# B&R Automation Studio project CombinedLinenSoiledA9KAN (part 3)

#### 6_sdc1Cyclic.ab
```automation-basic
PROGRAM _CYCLIC
	(* cyclic program *)

;Sequence 6 - Discharger 1 D[906]
a

;-----------------------------------------
;Revision 1.00 19/12/2005 D.J. First Issue
;-----------------------------------------

DischargerEnable 		= ((D[17] > 0) AND NOT Std.HaltSys)

I_BagAtBuffer			  = X[3].X06
I_BagAtDischarger	= X[3].X05
I_BagEmpty        = X[6].X01

I_OpenBag				= CAN[2].DropLoad OR TestDrop           ;X[23].X01
I_LoadDropped			= CAN[2].LoadDropped OR TestDischarger  ;X[23].X02

O_Steadys				= FALSE ;Y[6].Y01
O_OpenBuffer 			= FALSE ;Y[6].Y02
O_OpenBag				= FALSE ;Y[6].Y03
O_OpenStop				= FALSE ;Y[6].Y04
O_Closer				= FALSE ;Y[6].Y05

;Alarm
Alarm[7].Name 			= 0 ;Clear sequence alarm name
Alarm[7].Bag 			= 231
Alarm[7].Beacon			= TRUE
Alarm[7].Extra			= 0
Alarm[7].Time			= 3000

;Setup Sequence
STEP = D[907]
;Setup Pulse contact
PLS = (STEP <> LASTSTEP)
LASTSTEP = STEP

;Step 0 - Disabled
IF (STEP = 0) THEN
	;Disabled
ENDIF

;Check Status - Bag settled at buffer, no bag at discharger, bag at buffer on screen and no bag at discharger on the screen
TON_10ms(I_BagAtBuffer,300,SettledAtBuffer,SettledAtBufferET)
IF (STEP = 1) THEN
	IF (DischargerEnable AND SettledAtBuffer AND NOT I_BagAtDischarger AND (Bag[231].Cat = 0) AND NOT Std.HaltSys) THEN
		D[907] = 2
	ENDIF
	IF (Bag[231].Cat > 0) THEN
		Alarm[7].Name = almBagDataError
	ELSE IF I_BagAtDischarger THEN
		Alarm[7].Name = almSwitchFault
	ENDIF
ENDIF

;Wait for bag in discharger
IF (STEP = 2) THEN
	O_OpenBuffer 	= TRUE
	;Enable.SDC[1] 	= TRUE
	IF I_BagAtDischarger THEN
		D[907] = 3
	ENDIF
	Alarm[7].Name = almBagNotArrived
ENDIF

;Let bag settle in discharger
TON_10ms(((STEP = 3) AND I_BagAtDischarger),1000,SettledAtDischarger,SettledAtDischargerET)
IF (STEP = 3) THEN
	IF (Bag[231].Cat = 0) AND (Bag[229].Cat > 0) THEN
		Bag[231] = Bag[229]
		Bag[229] = Bag[0]
	ENDIF
	IF SettledAtDischarger THEN
		D[907] = 4
	ENDIF
	Alarm[7].Name = almBagNotSettled
ENDIF

;Allow steadys to move down
TON_10ms((STEP = 4),400,SteadysDown,SteadysDownET)
IF (STEP = 4) THEN
	IF SteadysDown AND (Bag[231].Cat <> Std.MaxCats)  THEN
		D[907] = 5
	ENDIF
	IF (Bag[231].Cat = Std.MaxCats) AND SteadysDown THEN
		D[907] = 10
	ENDIF
ENDIF

;Steady cylinders on from steps 4 - 9
O_Steadys = ((STEP >= 4) AND (STEP <= 9))

;Bag opener on from step 5 - 8
O_OpenBag = ((STEP >= 6) AND (STEP <= 8))

;Wash Codes
IF (STEP = 4) OR (STEP = 5) THEN

;round up weight to give to wash machine
	Remainder = SINT(Bag[231].Wgt MOD 10)
	IF (Remainder > 4) THEN
		WgtRound = (Bag[231].Wgt + 10)
	ELSE
		WgtRound = Bag[231].Wgt
	ENDIF

;Codes to CBW
	CAN[2].Category = Bag[231].Cat
	CAN[2].Customer = Bag[231].Cus
	CAN[2].Weight   = (WgtRound / 10)
ELSE
	CAN[2].Category = 0
	CAN[2].Customer = 0
	CAN[2].Weight   = 0
ENDIF

;Bag Ready to Washing Machine
IF (STEP = 5) THEN
	CAN[2].BagReady = TRUE
	IF I_OpenBag OR TestDischarger THEN
		D[907] = 6
	ENDIF
ELSE
	CAN[2].BagReady = FALSE
ENDIF

;Set LoadDropped to False
IF (STEP <> 6) THEN
	LoadDropped = FALSE
ENDIF

;Open Bag Until LoadDropped recieved and has been open for 6 seconds
TON_10ms((STEP = 6),600,MinOpen,MinOpenET) ;ET means Elapsed Time
IF (STEP = 6) THEN

	IF I_LoadDropped OR TestDischarger THEN
	;IF I_BagEmpty THEN
		LoadDropped = TRUE
	ENDIF

	IF (LoadDropped AND MinOpen) THEN
		;Write Report
		;------------
		IF (ReportUnloading[1].Cat = 0) THEN
			ReportUnloading[2].Cat = UINT(Bag[231].Cat)	;Category
			ReportUnloading[2].Cus = UINT(Bag[231].Cus)   ;Customer
			ReportUnloading[2].Wgt = Bag[231].Wgt		;Weight
			ReportUnloading[2].Cnt = 0					;Count
			ReportUnloading[2].Stn = 0					;Station
			ReportUnloading[2].Mcn = 2					;Machine
			;Bag[201]               = Bag[120]           ;move bag into machine tracking
		ENDIF
	ENDIF
	IF (LoadDropped AND MinOpen) THEN
		D[907] = 7
	ENDIF
	Alarm[7].Name = almLoadNotDropped
ENDIF

;Change display to empty bag
IF (STEP = 7) THEN
	IF ((NOT I_OpenBag AND NOT I_LoadDropped OR TestDrop)) THEN ;AND I_BagEmpty) OR TestDrop) THEN
		Bag[231].Cat 	= Std.MaxCats
		D[907] 			= 8
	ENDIF
	Alarm[7].Name = almGeneralSequence
ENDIF

;Close bag
TON_10ms((STEP = 8),700,CloserDown,CloserDownET)
IF (STEP = 8) THEN
	O_Closer = TRUE
	IF CloserDown THEN
		D[907] = 9
	ENDIF
ENDIF

;Allow closer to go back up
TON_10ms((STEP = 9),700,CloserUp,CloserUpET)
IF (STEP = 9) THEN
	IF CloserUp THEN
		D[907] = 10
	ENDIF
ENDIF

;Allow steadys to go up
TON_10ms((STEP = 10),400,SteadyUp,SteadyUpET)
IF (STEP = 10) THEN
	IF SteadyUp THEN
		D[907] = 11
	ENDIF
ENDIF

;Check for space on empty bag buffer
IF (STEP = 11) THEN
		Request.SDC[2] = TRUE
	IF Enable.SDC[2] THEN ;AND NOT I_BagAtEmptyBuffer AND NOT O_EmptyBagBufferOpen) THEN
		D[907] = 12
	ENDIF
	ELSE
			Request.SDC[2] = FALSE
ENDIF

;Open buffer stop - unitl bag out
IF (STEP = 12) THEN
	O_OpenStop = TRUE
	IF PLS THEN
		;C[14] = 0
	ENDIF
	Bag[231].Cat = 0
	Bag[231].Cus = 0
	Bag[231].Wgt = 0
	IF NOT Enable.SDC[2] THEN
		D[907] = 1
	ENDIF
	Alarm[7].Name = almBagNotReleased
ENDIF

;Alarms
TimerAlarm.IN 	= NOT PLS AND (Alarm[7].Name > 0)
TimerAlarm.PT 	= Alarm[7].Time
TimerAlarm FUB TON_10ms()
Alarm[7].On 	= TimerAlarm.Q
Alarm[7].ET 	= TimerAlarm.ET

;Outputs
Y[3].Y06 = O_OpenBuffer
Y[3].Y07 = O_Steadys
Y[3].Y08 = O_OpenBag
Y[3].Y09 = O_OpenStop
Y[3].Y10 = O_Closer

END_PROGRAM
```

### Program Logical/Sequences/10ms/8_svc1 (IEC) - * SVC1 Inverter VC

#### 7_svc1.var
```iecst
VAR RETAIN
	STEP : UINT;
END_VAR
VAR
	PLS : BOOL;
END_VAR
VAR RETAIN
	LASTSTEP : UINT;
END_VAR
VAR
	I_CarrAtTop : BOOL;
	I_BagOnCarr : BOOL;
	I_CarrAtBottom : BOOL;
	O_OpenCarrStop : BOOL;
	O_MoveCarrDown : BOOL;
	O_MoveCarrUp : BOOL;
	BagSettled : BOOL;
	O_OpenBufferStop : BOOL;
	BagAtBuffer : BOOL;
	MoveUpToFullOut : BOOL;
	MoveDownToBot : BOOL;
	Status : UINT;
	HighSpeedDoneET : TIME;
	I_BagBagReleased : BOOL;
	TONHighSpeed : TON_10ms;
	TimerAlarm : TON_10ms;
	HighSpeedTime : UINT;
	HighSpeedDone : BOOL;
	BagAtBufferET : TIME;
	I_BagAtBufferStop : BOOL;
	MoveDownEBagIn : BOOL;
	DDDDDD : BOOL;
	BagSettledET : TIME;
	I_CarriageAtTop : BOOL;
	I_CarriageAtBottom : BOOL;
	I_BagOnCarriage : BOOL;
	I_BagReleased : BOOL;
	O_MoveUp : BOOL;
	O_MoveDown : BOOL;
	O_OpenStop : BOOL;
	SettledOnCarriage : BOOL;
	SettledOnCarriageET : UDINT;
	E : BOOL;
	HighSpeedUp : BOOL;
	HighSpeedUpET : UDINT;
	HighSpeedDn : BOOL;
	HighSpeedDnET : UDINT;
END_VAR
```

#### 7_svc1Cyclic.ab
```automation-basic
PROGRAM _CYCLIC
	(* cyclic program *)
DDDDDD

I_CarriageAtTop			= X[3].X09
I_CarriageAtBottom		= X[3].X10
I_BagOnCarriage			= X[3].X11
I_BagReleased 			= X[3].X12

O_MoveUp 				= FALSE
O_MoveDown 				= FALSE
O_OpenStop 				= FALSE

Request.SVC[1] 			= FALSE
Enable.SLU1	 			= FALSE

;Setup Sequence
;-----------------------
STEP = D[908]
;Setup Pulse contact
PLS = (STEP <> LASTSTEP)
LASTSTEP = STEP

;Alarm
Alarm[8].Name 		= 0
Alarm[8].Bag		= 221
Alarm[8].Beacon		= TRUE
Alarm[8].Extra	 	= 0
Alarm[8].Time		= 3000
;Step 0 - Disabled
IF (STEP = 0) THEN
	;Disabled
ENDIF

;Wait for bag on carriage
IF (STEP = 1) THEN
	Enable.SLU1 = (I_CarriageAtBottom AND (NOT I_BagOnCarriage))
	IF I_BagOnCarriage THEN
		;BAGMOVE2(I_BagOnCarriage,mem_adr_E,220,221,BagSpacing)
			IF (Bag[220].Cat>0) AND (Bag[221].Cat=0) THEN
						Bag[221] = Bag[220]
						Bag[220] = Bag[0]
			ENDIF
		D[908] = 2
	ENDIF
ENDIF

IF (STEP = 2) THEN
	D[908] = 3
ENDIF

;Bag settles on carriage
TON_10ms(I_BagOnCarriage,300,SettledOnCarriage,SettledOnCarriageET)
IF (STEP = 3) THEN
	IF SettledOnCarriage THEN
		D[908] = 4
	ENDIF
ENDIF

;Move carriage up to top
IF (STEP = 4) THEN
	O_MoveUp = (NOT I_CarriageAtTop)
	IF I_CarriageAtTop THEN
		D[908] = 5
	ENDIF
ENDIF

;Check for space at SIC1 Buffer
IF (STEP = 5) THEN
	IF (Line[15].Clear AND NOT Y[5].Y14 AND (Bag[222].Cat = 0) AND (Bag[223].Cat = 0) AND NOT I_BagReleased) THEN
		D[908] = 6
	ENDIF
ENDIF

;Release bag, high-level
IF (STEP = 6) THEN
	O_OpenStop = I_CarriageAtTop
	;BAGMOVE2(PLS,mem_adr_E,221,222,BagSpacing)
	IF (Bag[221].Cat>0) AND (Bag[222].Cat=0) THEN
						Bag[222] = Bag[221]
						Bag[221] = Bag[0]
			ENDIF
	IF PLS THEN
		C[15] = 0	;Reset Trip Count
	ENDIF

	IF NOT PLS AND (C[15] > 0) THEN
		D[908] = 7
	ENDIF
ENDIF

;Move carriage down to Bottom
IF (STEP = 7) THEN
	IF I_BagOnCarriage THEN
				D[908] = 20
	ENDIF
	O_MoveDown = (NOT I_CarriageAtBottom)
	IF I_CarriageAtBottom THEN
		D[908] = 1
	ENDIF
ENDIF

 IF (STEP = 20) THEN
	Alarm[8].Name 		= almSwitchFault
	Alarm[8].Time		= 3
ENDIF

;Bag in transit to SIC1 buffer
IF ((Bag[222].Cat> 0) AND Line[15].Full) THEN
	;BAGMOVE2(TRUE,mem_adr_E,222,223,BagSpacing)
		IF (Bag[222].Cat>0) AND (Bag[223].Cat=0) THEN
						Bag[223] = Bag[222]
						Bag[222] = Bag[0]
			ENDIF
ENDIF

;Inverter Speed Selections
;-------------------------
;High Speed Used For Up		= 60Hz
;Medium Speed Used For Down	= 80Hz

;Alarms
TimerAlarm.IN = NOT PLS AND (Alarm[8].Name > 0)
TimerAlarm.PT = Alarm[8].Time
TimerAlarm FUB TON_10ms()
Alarm[8].On = TimerAlarm.Q
Alarm[8].ET = TimerAlarm.ET

TON_10ms(O_MoveUp  ,1680,HighSpeedUp,HighSpeedUpET) 	;Expected 16.94 seconds @ 591mm/sec
TON_10ms(O_MoveDown,1630,HighSpeedDn,HighSpeedDnET) 		;Expected 16.94 seconds @ 591mm/sec
IF (STEP = 4) THEN
	Y[9].Y01 = (NOT HighSpeedUp) 							;High Speed
	Y[9].Y02 = FALSE										;Medium Speed
ELSE IF (STEP = 7) THEN
	Y[9].Y01 = FALSE										;High Speed
	Y[9].Y02 = (NOT HighSpeedDn)							;Medium Speed
ELSE
	Y[9].Y01 = FALSE
	Y[9].Y02 = FALSE
ENDIF

;PLC Outputs
;-----------
Y[10].Y01 = O_MoveUp
Y[10].Y02 = O_MoveDown
Y[10].Y03 = (O_MoveUp OR O_MoveDown)
Y[10].Y04 = O_OpenStop

;Inverter Parameters
;2	Min Freq			20Hz
;4	High Speed			60Hz
;5	Medium Speed		80Hz
;7  Acceleration Time	0.5sec
;8  Deceleration Time	0.5sec
;9  Electronic O/L		5.00A
;10	DC Injection freq	7Hz
;11 DC Injection Time	1sec
;12	DC Brake Voltage	14%
;13	Starting freq		20Hz
;30	Regenerative fun	1
;42	Output freq detect	0.5Hz
;70	Brake duty			5%
;79 Operation mode		3
;80 Motor capicity 		1.5Kw
;83	Rated motor voltage	400v
;84	Rated motor freq	50Hz
END_PROGRAM
```

### Program Logical/Sequences/10ms/9_sic1 (IEC, version 1.00.0) - * SPC1 Empty bags up

#### 9_spc1Cyclic.ab
```automation-basic
PROGRAM _CYCLIC
	(* cyclic program *)

;----------------------------------------------
;Sequence 10 - SPC1 Pneumatic Conveyor 1 D[910]
;----------------------------------------------

;Inputs
;Incline Conveyor
;-----------------------------------------
;Revision 1.00 09/01/2002 D.J. First Issue
;-----------------------------------------

I_PaddleinPosition		= X[5].X08
I_BaginIncline			= X[5].X07
I_BagatBuffer			= X[5].X10

O_RunMotor 				= FALSE
O_OpenBufferStop		= FALSE

Request.SIC[1]			= FALSE

;Setup Sequence
;-----------------------
STEP = D[909]
;Setup Pulse contact
PLS = (STEP <> LASTSTEP)
LASTSTEP = STEP

Alarm[9].Name 		= 0
Alarm[9].Bag		= 224
Alarm[9].Beacon		= TRUE
Alarm[9].Extra	 	= 0
Alarm[9].Time		= 3000
;Alarm
;TON_10ms(((NOT PLS) AND (STEP = 3)),1000,Alarm[9],AlarmET[9])

;Run Incline until paddle in position
IF (STEP = 1) THEN
	O_RunMotor = (NOT I_PaddleinPosition)
	IF I_PaddleinPosition THEN
		D[909] = 2
	ENDIF
	Alarm[9].Name 		= almSwitchFault
ENDIF

;Check romm in buffer
TON_10ms(I_BagatBuffer,300,BagSettledBuffer,BagSettledBufferET)
IF (STEP = 2) THEN
	IF (BagSettledBuffer AND (Bag[224].Cat = 0)) THEN
		D[909] = 3
	ENDIF
ENDIF

;Open Stop on steps 3 - 5
IF (STEP >= 3) AND (STEP <= 5) THEN
	O_OpenBufferStop = TRUE
ENDIF

;Wait for bag in incline
IF (STEP = 3) THEN
	;BAGMOVE2(PLS,mem_adr_E,223,224,BagSpacing)
	IF (Bag[223].Cat>0)AND (Bag[224].Cat=0)THEN
				Bag[224] = Bag[223]
				Bag[223] = Bag[0]
	ENDIF
	IF I_BaginIncline THEN
		D[909] = 4
	ENDIF
	Alarm[9].Name 		= almBagNotReleased
ENDIF

;Let bag settle at base of incline
TON_10ms((STEP = 4),300,BagSettled,BagSettledET)
IF (STEP = 4) THEN
	IF BagSettled THEN
		D[909] = 5
	ENDIF
ENDIF

;Move Bag up incline
TON_10ms((STEP = 5),200,BagNearTop,BagNearTopET)
IF (STEP = 5) THEN
	O_RunMotor = TRUE
	IF BagNearTop THEN
		D[909] = 6
	ENDIF
ENDIF

;Wait for Ongoing Sequence to Enable
;Run motor for 0.5 seconds
TON_10ms((STEP = 6),50,RunOn,RunOnET)
IF (STEP = 6) THEN
	O_RunMotor 		= NOT RunOn
	Request.SIC[1] 	= TRUE
	IF Enable.SIC[1] THEN
		D[909] = 7
	ENDIF
ENDIF

;Run incline until bag at storage lines
IF (STEP = 7) THEN
	;BAGMOVE2(PLS,mem_adr_E,224,225,BagSpacing)
	IF (Bag[224].Cat>0)AND (Bag[225].Cat=0)THEN
				Bag[225] = Bag[224]
				Bag[224] = Bag[0]
	ENDIF
	O_RunMotor = TRUE
	;Bag in transit arrives at the buffers
	IF NOT Enable.SIC[1] THEN
		D[909] = 1
	ENDIF
	Alarm[9].Name 		= almBagNotReleased
ENDIF

;Alarms
TimerAlarm.IN = NOT PLS AND (Alarm[9].Name > 0)
TimerAlarm.PT = Alarm[9].Time
TimerAlarm FUB TON_10ms()
Alarm[9].On = TimerAlarm.Q
Alarm[9].ET = TimerAlarm.ET

Y[10].Y09 = O_RunMotor
Y[5].Y14 = O_OpenBufferStop
END_PROGRAM
```

#### 9_spc1.var
```iecst
VAR
	I_CarrAtTop : BOOL;
	I_CarrAtBottom : BOOL;
END_VAR
VAR RETAIN
	STEP : UINT;
END_VAR
VAR
	PLS : BOOL;
END_VAR
VAR RETAIN
	LASTSTEP : UINT;
END_VAR
VAR
	O_MoveCarrUp : BOOL;
	O_OpenCarrStop : BOOL;
	O_MoveCarrDown : BOOL;
	I_BagOnCarr : BOOL;
	O_OpenBuffer : BOOL;
	SettledBuffer : BOOL;
	SettledBufferET : TIME;
	I_BagAtBuffer : BOOL;
	BagSettledOnCarr : BOOL;
	BagSettledOnCarrET : TIME;
	I_BagReleased : BOOL;
	TimerAlarm : TON_10ms;
	I_BagAtLLBuff : BOOL;
	O_LLBuffOpen : BOOL;
	SettledBufferSDC2ET : TIME;
	SettledBufferSDC2 : BOOL;
	I_BagAtBufferSDC2 : BOOL;
	Alt : USINT;
	O_OpenBuffer1 : BOOL;
	I_PaddleinPosition : BOOL;
	I_BaginIncline : BOOL;
	I_BagatBuffer : BOOL;
	O_RunMotor : BOOL;
	O_OpenBufferStop : BOOL;
	BagSettledBuffer : BOOL;
	BagSettledBufferET : UDINT;
	BagSettled : BOOL;
	BagSettledET : UDINT;
	BagNearTop : BOOL;
	BagNearTopET : UDINT;
	RunOn : BOOL;
	RunOnET : UDINT;
END_VAR
```

### Program Logical/Sequences/10ms/10_bson (IEC) - * SBSN1 Bagstacker Ongoing 

#### 10_bson.var
```iecst
VAR
	I_OnLineA : BOOL;
	I_TiltA : BOOL;
	I_TiltB : BOOL;
	I_Bagout : BOOL;
	O_OpenBufferStop : BOOL;
	O_SelectLineA : BOOL;
	O_SelectLineB : BOOL;
	O_OpenStops : BOOL;
	O_TiltCylinder : BOOL;
	O_OperatePusher : BOOL;
	PLS : BOOL;
END_VAR
VAR RETAIN
	LASTSTEP : UINT;
	STEP : UINT;
END_VAR
VAR
	TiltDownET : UDINT;
	TiltDown : BOOL;
	TiltUpET : UDINT;
	TiltUp : BOOL;
	NotFullET : UDINT;
	NotFull : BOOL;
	RequirePusherET : UDINT;
	Pushed : BOOL;
	PushedET : UDINT;
	BagAtTiltET : TIME;
	BagAtTilt : BOOL;
	PointReset : BOOL;
	PointResetET : TIME;
	TimerAlarm : TON_10ms;
	ResetPoint : BOOL;
	ResetPointET : UDINT;
	BagatTilt : BOOL;
	BagatTiltET : UDINT;
	PR1_LineClearET : UDINT;
	PR2_LineClearET : UDINT;
	PR3_LineClearET : UDINT;
	PR4_LineClearET : UDINT;
END_VAR
```

#### 10_bsonCyclic.ab
```automation-basic
PROGRAM _CYCLIC
(* cyclic program *)

;----------------------------------------
;Sequence 14 - Ongoing Bag Stacker D[910]
;----------------------------------------

;Inputs
I_TiltA					= X[6].X02
I_TiltB					= X[6].X03
I_OnLineA		  		= X[6].X04
I_Bagout				= X[6].X05

O_SelectLineA			= FALSE
O_SelectLineB			= FALSE
O_OperatePusher			= FALSE
O_TiltCylinder			= FALSE
O_OpenStops				= FALSE
O_OpenBufferStop		= FALSE

;Setup Sequence
;-----------------------
STEP = D[910]
;Setup Pulse contact
PLS = (STEP <> LASTSTEP)
LASTSTEP = STEP

;Alarm
Alarm[10].Name 		= 0
Alarm[10].Bag		= 10003
Alarm[10].Beacon		= TRUE
Alarm[10].Extra	 	= 0
Alarm[10].Time		= 3000

IF (STEP = 0) THEN
	;Do Nothing
ENDIF

;Select Line 'a'
TON_10ms((STEP = 1),100,ResetPoint,ResetPointET)
IF (STEP = 1) THEN
	O_SelectLineA = TRUE
	IF ResetPoint AND (D[22]>0)THEN
		D[910] = 2
	ENDIF
ENDIF

;Wait for bag to be ready
IF (STEP = 2) THEN
	IF (Request.SDC[1] OR Request.SDC[2]) THEN
		D[910] = 3
	ENDIF
ENDIF

;Enable requesting discharger to send a bag
IF (STEP = 3) THEN
	IF I_OnLineA THEN
		D[910] = 4
	ELSE
		;Set Bags from SDC1 or SDC1
		IF (Request.SDC[1] AND NOT Enable.SDC[2]) THEN
			Enable.SDC[1] = TRUE
		ELSE IF (Request.SDC[2] AND NOT Enable.SDC[1]) THEN
			Enable.SDC[2] = TRUE
		ENDIF
	ENDIF
ELSE
	Enable.SDC[1] = FALSE
	Enable.SDC[2] = FALSE
ENDIF

;Wait for bag in Tilt position
TON_10ms((I_TiltA AND I_TiltB),300,BagatTilt,BagatTiltET)
IF (STEP = 4) THEN
	O_SelectLineB = TRUE
	IF BagatTilt THEN
		D[910] = 5
	ENDIF
ENDIF

;Tilt down
TON_10ms((STEP = 5),500,TiltDown,TiltDownET)
IF (STEP = 5) THEN
	O_TiltCylinder = TRUE
	IF TiltDown THEN
		D[910] = 6
	ENDIF
ENDIF

;Tilt up
TON_10ms((STEP = 6),500,TiltUp,TiltUpET)
IF (STEP = 6) THEN
	IF TiltUp THEN
		D[910] = 7
	ENDIF
ENDIF

;Check not full
TON_10ms((NOT I_Bagout),300,NotFull,NotFullET)
IF (STEP = 7) THEN
	IF NotFull THEN
		D[910] = 8
	ENDIF
ENDIF

;Open stops to release bag
IF (STEP = 8) THEN
	O_OpenStops = TRUE
	IF I_Bagout THEN
		D[910] = 1
	ENDIF
ENDIF

;Pusher Cylinder
TON_10ms(((STEP = 7) OR (STEP = 8)) AND (NOT Pushed),500,O_OperatePusher,RequirePusherET)
TON_10ms(O_OperatePusher,500,Pushed,PushedET)

;Bagstacker Pressure relief 1
TON_10ms((NOT X[6].X06) AND (NOT X[6].X07),500,Y[6].Y06,PR1_LineClearET)

;Bagstacker Pressure relief 2
TON_10ms((NOT X[7].X03) AND (NOT X[7].X04),500,Y[6].Y15,PR2_LineClearET)

;Bagstacker Pressure relief 3
TON_10ms((NOT X[7].X01) AND (NOT X[7].X02),500,Y[7].Y01,PR3_LineClearET)

;Bagstacker Pressure relief 4 - Offgoing
TON_10ms((NOT X[6].X14) AND (NOT X[6].X15),500,Y[6].Y14,PR4_LineClearET)

;Alarms
TimerAlarm.IN = NOT PLS AND (Alarm[10].Name > 0)
TimerAlarm.PT = Alarm[10].Time
TimerAlarm FUB TON_10ms()
Alarm[10].On = TimerAlarm.Q
Alarm[10].ET = TimerAlarm.ET

Y[5].Y10 = Enable.SDC[2]
Y[5].Y11 = Enable.SDC[1]

Y[6].Y01 = O_SelectLineA
Y[6].Y02 = O_SelectLineB
Y[6].Y03 = O_OpenStops
Y[6].Y04 = O_OperatePusher
Y[6].Y05 = O_TiltCylinder

END_PROGRAM
```

### Program Logical/Sequences/10ms/11_bsoff (IEC, version 1.00.0) - * SBSF1 Bagstacker Offgoing

#### 11_bsoffCyclic.ab
```automation-basic
PROGRAM _CYCLIC
  	(* cyclic program *)

;-----------------------------------------
;Sequence 11 - Offgoing Bag Stacker D[911]
;-----------------------------------------

;Inputs
I_LevelA				= X[6].X10
I_LevelB				= X[6].X11
I_RockSepA				= X[6].X08
I_RockSepB				= X[6].X09
I_OutLineA				= X[6].X12
I_AtRotary				= X[6].X13

;O_SelectLineA			= FALSE
;O_SelectLineB			= FALSE
O_RotatePoint			= FALSE
O_OpenRockSep			= FALSE
O_OpenLineAStop			= FALSE
O_OpenLineBStop			= FALSE
O_LevelCylinder			= FALSE
O_OpenRotaryPoint		= FALSE

;Setup Sequence
;-----------------------
STEP = D[911]
;Setup Pulse contact
PLS = (STEP <> LASTSTEP)
LASTSTEP = STEP

;Alarm
Alarm[11].Name 		= 0
Alarm[11].Bag		= 10002
Alarm[11].Beacon		= TRUE
Alarm[11].Extra	 	= 0
Alarm[11].Time		= 3000

;Select Line 'A'
TON_10ms((STEP = 1) AND ((NOT I_LevelA) AND (NOT I_LevelB)),100,SelectA,SelectAET)
IF (STEP = 1) THEN
	;O_SelectLineA = TRUE
	IF SelectA THEN
		D[911] = 2
	ENDIF
ENDIF

;Open seperators wait for leveller to be ready
TON_10ms(((STEP = 2) AND I_RockSepA AND I_RockSepB),200,RockerReady,RockerReadyET)
IF (STEP = 2) THEN
	O_OpenRockSep = (STEP = 2)
	IF RockerReady THEN
		D[911] = 3
	ENDIF
ENDIF

;Wait for bag to be in leveller position
TON_10ms((I_LevelA AND I_LevelB),400,LevellerFull,LevellerFullET)
IF (STEP = 3) THEN
	IF LevellerFull THEN
		D[911] = 4
	ENDIF
ENDIF

;Move bag leveller down
TON_10ms((STEP = 4),500,LevellerDown,LevellerDownET)
IF (STEP = 4) THEN
	O_LevelCylinder = TRUE
	IF LevellerDown THEN
		D[911] = 5
	ENDIF
ENDIF

;Allow bag leveller to retract
TON_10ms((STEP = 5),500,LevellerUp,LevellerUpET)
IF (STEP = 5) THEN
	IF LevellerUp THEN
		D[911] = 6
	ENDIF
ENDIF

;Check romm in buffer
IF (STEP = 6) THEN
	IF (Line[16].Clear AND NOT Y[3].Y16) THEN
		D[911] = 7
	ENDIF
ENDIF

;Open stop on line 'A'
IF (STEP = 7) THEN
	O_OpenLineAStop = TRUE
	IF PLS THEN
		C[16] = 0
	ENDIF
	IF I_OutLineA THEN
		D[911] = 8
	ENDIF
ENDIF

;Open stop on line 'B'until bag in rotary point
TON_10ms(I_AtRotary,300,SettledInRotary,SettledInRotaryET)
IF (STEP = 8) THEN
	O_OpenLineBStop = TRUE
	IF SettledInRotary THEN
		D[911] = 9
	ENDIF
ENDIF

;Select bag stop and wait for bag out of leveller
TON_10ms((STEP = 9),300,PointRotated,PointRotatedET)
IF (STEP = 9) THEN
	O_OpenLineBStop 	= TRUE
	O_RotatePoint 		= TRUE
	O_OpenRotaryPoint 	= PointRotated
	IF Line[16].Full THEN
		D[911] = 1
	ENDIF
ENDIF

;Alarms
TimerAlarm.IN = NOT PLS AND (Alarm[11].Name > 0)
TimerAlarm.PT = Alarm[11].Time
TimerAlarm FUB TON_10ms()
Alarm[11].On = TimerAlarm.Q
Alarm[11].ET = TimerAlarm.ET

;Y000 = O_SelectLineA
;Y000 = O_SelectLineB
Y[6].Y12 = NOT O_RotatePoint
Y[6].Y13 = O_OpenRotaryPoint
Y[6].Y10 = O_OpenRockSep
Y[6].Y08 = O_OpenLineAStop
Y[6].Y09 = O_OpenLineBStop
Y[6].Y11 = O_LevelCylinder
END_PROGRAM
```

#### 11_bsoff.var
```iecst
VAR RETAIN
	STEP : UINT;
END_VAR
VAR
	PLS : BOOL;
END_VAR
VAR RETAIN
	LASTSTEP : UINT;
END_VAR
VAR
	LevellerDownET : TIME;
	O_LevelCylinder : BOOL;
	O_SelectLineB : BOOL;
	O_SelectLineA : BOOL;
	I_OutLineB : BOOL;
	LevellerDown : BOOL;
	LevellerUp : BOOL;
	LevellerUpET : TIME;
	I_TiltB : BOOL; (* SPR1 Trolley past stop *)
	I_OutLineA : BOOL;
	O_OpenRockSep : BOOL;
	O_OpenLineAStop : BOOL;
	O_OpenLineBStop : BOOL;
	I_RockSepA : BOOL;
	I_RockSepB : BOOL;
	I_TiltA : BOOL; (* SBS1 ON Bag on stacker *)
	O_LevelCylinderUP : BOOL;
	PRLineClearET : ARRAY[0..4] OF TIME;
	SettledLevel : BOOL;
	SettledLevelET : TIME;
	SettledInSepsET : TIME;
	SettledInSeps : BOOL;
	LevelClearET : TIME;
	LevelClear : BOOL;
	TimerAlarm : TON_10ms;
	I_LevelA : BOOL;
	I_LevelB : BOOL;
	I_AtRotary : BOOL;
	O_RotatePoint : BOOL;
	O_OpenRotaryPoint : BOOL;
	AlarmET : UDINT;
	SelectA : BOOL;
	SelectAET : UDINT;
	RockerReady : BOOL;
	RockerReadyET : UDINT;
	LevellerFull : BOOL;
	LevellerFullET : UDINT;
	SettledInRotary : BOOL;
	SettledInRotaryET : UDINT;
	PointRotated : BOOL;
	PointRotatedET : UDINT;
END_VAR
```

### Program Logical/Sequences/10ms/12_svc2 (IEC) - * SVC2 2-level - Inverter

#### 12_svc2.var
```iecst
VAR
	I_CarrAtTop : BOOL;
	I_CarrAtBottom : BOOL;
END_VAR
VAR RETAIN
	STEP : UINT;
END_VAR
VAR
	PLS : BOOL;
END_VAR
VAR RETAIN
	LASTSTEP : UINT;
END_VAR
VAR
	O_MoveCarrUp : BOOL;
	O_OpenCarrStop : BOOL;
	O_MoveCarrDown : BOOL;
	I_BagOnCarr : BOOL;
	Speed1 : BOOL;
	MoveDownToBot : BOOL;
	Speed2 : BOOL;
	O_SelectSP1 : BOOL;
	MoveUpToFullOut : BOOL;
	I_BagReleased : BOOL;
	TimerAlarm : TON_10ms;
	I_CarrAtEBagOut : BOOL;
	O_SelectPoint : BOOL;
	O_OpenFullBuffer : BOOL;
	HighSpeedDone : BOOL;
	HighSpeedTime : UDINT;
	TONHighSpeed : TON_10ms;
	MoveDownEBagIn : BOOL;
	HighSpeedDoneET : TIME;
	SettledAtBuffer : BOOL;
	SettledAtBufferET : TIME;
	I_CarriageAtTop : BOOL;
	I_CarriageAtBottom : BOOL;
	I_BagOnCarriage : BOOL;
	I_BagAtBuffer : BOOL;
	O_MoveUp : BOOL;
	O_MoveDown : BOOL;
	O_OpenStop : BOOL;
	O_OpenBufferStop : BOOL;
	EBagReady : BOOL;
	EBagReadyET : UDINT;
	BagSettled : BOOL;
	BagSettledET : UDINT;
	HighSpeedUp : BOOL;
	HighSpeedUpET : UDINT;
	HighSpeedDn : BOOL;
	HighSpeedDnET : UDINT;
END_VAR
```

#### 12_svc2Cyclic.ab
```automation-basic
PROGRAM _CYCLIC
	(* cyclic program *)

;--------------------------------------------
;Sequence 8 - SVC1 Vertical conveyor 1 D[908]
;--------------------------------------------

;Inputs
I_CarriageAtTop			= X[3].X13
I_CarriageAtBottom		= X[3].X14
I_BagOnCarriage			= X[3].X15
I_BagAtBuffer			= X[3].X16

O_MoveUp 				= FALSE
O_MoveDown 				= FALSE
O_OpenStop 				= FALSE
O_OpenBufferStop		= FALSE

;Setup Sequence
;-----------------------
STEP = D[912]
;Setup Pulse contact
PLS = (STEP <> LASTSTEP)
LASTSTEP = STEP

IF (STEP = 7) AND I_BagOnCarriage THEN
	D[912]  = 20
ENDIF
;Alarm
Alarm[12].Name 		= 0
Alarm[12].Bag		= 10004
Alarm[12].Beacon		= TRUE
Alarm[12].Extra	 	= 0
Alarm[12].Time		= 3000

;Wait for Empty bag to be ready
TON_10ms(I_BagAtBuffer,300,EBagReady,EBagReadyET)
IF (STEP = 1) THEN
	IF EBagReady THEN
		D[912] = 2
	ENDIF
ENDIF

;Wait for bag on carriage
IF (STEP = 2) THEN
	O_OpenBufferStop = (I_CarriageAtTop AND (NOT I_BagOnCarriage))
	IF I_BagOnCarriage THEN
		D[912] = 3
	ENDIF
ENDIF

;Wait for bag to settle on carriage
TON_10ms(((STEP = 3) AND I_BagOnCarriage),300,BagSettled,BagSettledET)
IF (STEP = 3) THEN
	IF BagSettled THEN
		D[912] = 4
	ENDIF
ENDIF

;Move Carriage down to bottom
IF (STEP = 4) THEN
	O_MoveDown = (NOT I_CarriageAtBottom)
	IF I_CarriageAtBottom THEN
		D[912] = 5
	ENDIF
ENDIF

;Check if space available
;TON_10ms(((NOT Y711) AND (NOT X712)),200,SpaceEmpty,SpaceEmptyET)
IF (STEP = 5) THEN
	IF Enable.SVC2 THEN
		D[912] = 6
	ENDIF
ENDIF

;Open stop, let bag in buffer
IF (STEP = 6) THEN
	O_OpenStop = I_CarriageAtBottom
	;IF PLS THEN
	;	C[20] = 0
	;ENDIF
	IF NOT Enable.SVC2 THEN
		D[912] = 7
	ENDIF
ENDIF

;Move Carriage up to top
IF (STEP = 7) THEN
	O_MoveUp = (NOT I_CarriageAtTop)
	IF I_CarriageAtTop THEN
		D[912] = 1
	ENDIF
ENDIF

 IF (STEP = 20) THEN
	Alarm[12].Name 		= almSwitchFault
	Alarm[12].Time		= 3
ENDIF
;Inverter Speed Selections
;-------------------------
;High Speed Used For Up		= 60Hz
;Medium Speed Used For Down	= 60Hz

TON_10ms(O_MoveUp  ,920,HighSpeedUp,HighSpeedUpET) 	;Expected 16.94 seconds @ 591mm/sec
TON_10ms(O_MoveDown,900,HighSpeedDn,HighSpeedDnET) 		;Expected 16.94 seconds @ 591mm/sec
IF (STEP = 4) THEN
	Y[9].Y03 = (NOT HighSpeedDn) 							;High Speed
	Y[9].Y04 = FALSE										;Medium Speed
ELSE IF (STEP = 7) THEN
	Y[9].Y03 = FALSE										;High Speed
	Y[9].Y04 = (NOT HighSpeedUp)							;Medium Speed
ELSE
	Y[9].Y03 = FALSE
	Y[9].Y04 = FALSE
ENDIF

;Alarms
TimerAlarm.IN = NOT PLS AND (Alarm[12].Name > 0)
TimerAlarm.PT = Alarm[12].Time
TimerAlarm FUB TON_10ms()
Alarm[12].On = TimerAlarm.Q
Alarm[12].ET = TimerAlarm.ET
;Outputs
;-------
Y[10].Y05 = O_MoveUp
Y[10].Y06 = O_MoveDown
Y[10].Y07 = (O_MoveUp OR O_MoveDown)
Y[10].Y08 = O_OpenStop
Y[3].Y16 = O_OpenBufferStop

;Inverter Parameters
;2	Min Freq			20Hz
;4	High Speed			60Hz
;5	Medium Speed		60Hz
;7  Acceleration Time	0.5sec
;8  Deceleration Time	0.5sec
;9  Electronic O/L		5.00A
;10	DC Injection freq	7Hz
;11 DC Injection Time	1sec
;12	DC Brake Voltage	14%
;13	Starting freq		20Hz
;30	Regenerative fun	1
;42	Output freq detect	0.5Hz
;70	Brake duty			5%
;79 Operation mode		3
;80 Motor capicity 		1.5Kw
;83	Rated motor voltage	400v
;84	Rated motor freq	50Hz
END_PROGRAM
```

### Program Logical/Sequences/10ms/zzAI2744 (IEC) - Weight 

#### zzAI2744.var
```iecst
(********************************************************************
 * COPYRIGHT -- Kannegiesser UK Ltd
 ********************************************************************
 * Program: zzAI2744
 * File: zzAI2744.var
 * Author: zmclaren
 * Created: May 25, 2012
 ********************************************************************
 * Local variables of program zzAI2744
 ********************************************************************)
VAR
	LastRawValue : ARRAY[0..59] OF DINT;
	i : USINT;
	NoChangeCounter : ARRAY[0..59] OF UINT;
END_VAR
```

### Program Logical/Sequences/10ms/ssr_sortbelt (IEC) - *Speed Reducers

#### p.var
```iecst
VAR
	myHaltSys : BOOL;
	O_CloseBrush : ARRAY[0..5] OF BOOL;
	I_BagApproach : ARRAY[0..5] OF BOOL;
	TON_OpenBrush : ARRAY[0..5] OF TON_10ms;
	n : USINT;
	myZone : INT;
	SettledAtSep : BOOL;
	O_OpenSep : BOOL;
	CloseSep : BOOL;
	I_BagAtRollerRockerBeforePDS1 : BOOL;
	SettledAtSepET : UDINT;
	CloseSepET : UDINT;
	I_BagAtBottom : BOOL;
END_VAR
```

#### p.ab
```automation-basic
;-------------
;Speed Reducer
;-------------

PROGRAM _INIT

END_PROGRAM
PROGRAM _CYCLIC

myZone					= 0
;myHaltSys				= Std.HaltSysZone[myZone]

;Sorting Belts
Y[5].Y15 = X[5].X15
Y[10].Y11 = X[5].X15
Y[10].Y12 = X[5].X15
Y[10].Y13 = X[5].X15
Y[10].Y14 = X[5].X15

LOOP n = 1 TO 5 DO
	IF I_BagApproach[n] THEN
		O_CloseBrush[n] = TRUE
	ENDIF
	TON_OpenBrush[n].IN = NOT myHaltSys AND O_CloseBrush[n]
	TON_OpenBrush[n].PT	= 300
	TON_OpenBrush[n] FUB TON_10ms()

	IF TON_OpenBrush[n].Q THEN
		O_CloseBrush[n] = FALSE
	ENDIF
ENDLOOP

TON_10ms(I_BagAtRollerRockerBeforePDS1 AND NOT O_OpenSep AND NOT I_BagAtBottom,200,SettledAtSep,SettledAtSepET)
TON_10ms(O_OpenSep,200,CloseSep,CloseSepET)
IF SettledAtSep THEN
	O_OpenSep = TRUE
ENDIF
IF CloseSep THEN
	O_OpenSep = FALSE
ENDIF

;Outputs
;Y[180].Y07		= O_CloseBrush[1]
;Y[122].Y07		= O_CloseBrush[2]
;Y[121].Y07		= O_CloseBrush[3]
;Y[121].Y08		= O_CloseBrush[4]
;Y[103].Y06		= O_CloseBrush[5]
;Y[178].Y07      = O_OpenSep
END_PROGRAM
```

### Program Logical/Sequences/10ms/zzIndi (IEC) - * Indication pictures on graphics

#### zzindiCyclic.ab
```automation-basic
PROGRAM _CYCLIC
(* cyclic program *)

;------------------------------
;Indication picture on graphics
;------------------------------

;-----------------------------------------
;Revision 1.00 19/10/2006 D.J. First Issue
;-----------------------------------------

;Write Indication[0 - 79] To D71 to D75

Offset = 0

LOOP n = 0 TO 4 DO

	Encode[n].Input[0] 	= Indication[0 + Offset]
	Encode[n].Input[1] 	= Indication[1 + Offset]
	Encode[n].Input[2] 	= Indication[2 + Offset]
	Encode[n].Input[3] 	= Indication[3 + Offset]
	Encode[n].Input[4] 	= Indication[4 + Offset]
	Encode[n].Input[5] 	= Indication[5 + Offset]
	Encode[n].Input[6] 	= Indication[6 + Offset]
	Encode[n].Input[7] 	= Indication[7 + Offset]
	Encode[n].Input[8] 	= Indication[8 + Offset]
	Encode[n].Input[9] 	= Indication[9 + Offset]
	Encode[n].Input[10] = Indication[10 + Offset]
	Encode[n].Input[11] = Indication[11 + Offset]
	Encode[n].Input[12] = Indication[12 + Offset]
	Encode[n].Input[13] = Indication[13 + Offset]
	Encode[n].Input[14] = Indication[14 + Offset]
	Encode[n].Input[15] = Indication[15 + Offset]

	Encode[n] FUB BIT_ENCODE()

	D[71 + n] = Encode[n].Output

	Offset = Offset + 16

ENDLOOP
END_PROGRAM
```

### Program Logical/Sequences/10ms/zzTCPIP (IEC) - * TCP IP Communications For Driver V5.0 and above

#### zztcpip.var
```iecst
VAR
	Port : UINT;
	IPAddr : UDINT;
	TCPsend_1 : TCPsend;
	TCPserv_1 : TCPserv;
	NoDataET : TIME;
	NoData : BOOL;
	PLS : BOOL;
	RXStatus : UINT;
	TCPclose_1 : TCPclose;
	RXLength : UDINT;
	NEWSTEP : UINT;
	STEP : UINT;
	TCPrecv_1 : TCPrecv;
	rdata : ARRAY[0..4999] OF USINT;
	Data_Array_Type : INT;
	Data_array_adr : UDINT;
	Data_StartH : UINT;
	Data_Start : UINT;
	Data_Amount : UINT;
	Data_Valid : BOOL;
	Data_RXTX_Type : INT;
	LengthValid : BOOL;
	tx_frame : ARRAY[0..4999] OF USINT;
	WriteEnable : BOOL;
	tx_length : UINT;
	RXValid : UINT;
	Data_AmountH : UINT;
	NEWSTEP2 : UINT;
	STEP2 : UINT;
	TCPserv_2 : TCPserv;
	Port2 : UINT;
	IPAddr2 : UDINT;
	PLS2 : BOOL;
	WriteEnable2 : BOOL;
	TCPsend_2 : TCPsend;
	TCPrecv_2 : TCPrecv;
	rdata2 : ARRAY[0..4999] OF USINT;
	RXLength2 : UDINT;
	RXStatus2 : UINT;
	RXValid2 : UINT;
	tx_frame2 : ARRAY[0..4999] OF USINT;
	tx_length2 : UINT;
	NoData2 : BOOL;
	NoData2ET : TIME;
	TCPclose_2 : TCPclose;
	PacketID : USINT;
	EnableConnection1 : BOOL;
	EnableConnection2 : BOOL;
	ResetConnection : BOOL;
	Bytes : UINT;
END_VAR
```

#### zztcpip.ab
```automation-basic
;-----------------------------------
;TCP IP Driver Communications Driver
;-----------------------------------

;------------------------------------------------------------------------------------------------------------
;Version 1.00 01/12/2005 D.J. First Issue
;Version 2.00 14/04/2009 D.J. Added VC_Posn data type
;Version 3.00 02/06/2009 D.J. Added D32 32-Bit Data
;Version 4.00 09/04/2010 D.J. Added MCN Machine Type Communication
;Version 4.10 03/11/2010 D.J. Changed VC to RB (Robo) other than that full compatiable with Version 4.00
;Version 5.00 28/04/2012 D.J. Enabled larger data size now 5000 bytes (200 bags with a size of 25 bytes each)
;------------------------------------------------------------------------------------------------------------

;Normally the driver will be sending constant requests - if the driver dosen't send anything for 1 second then the connection should be closed.

PROGRAM _INIT

;Enable connections set to TRUE or FALSE depending on how many connections are required
EnableConnection1 = TRUE
EnableConnection2 = TRUE

;Start Connection
ResetConnection = TRUE

END_PROGRAM

PROGRAM _CYCLIC

;------------
;Connection 1
;------------

;Restart - from init routine
IF ResetConnection THEN
	IF EnableConnection1 THEN
		NEWSTEP = 1
	ELSE
		NEWSTEP = 0
	ENDIF
ENDIF

STEP = NEWSTEP

;Disabled
IF STEP = 0 THEN
	;Do Nothing
ENDIF

;Init Server
IF STEP = 1 THEN
	TCPserv_1.enable = 1
	TCPserv_1.porta = 21001
	TCPserv_1 FUB TCPserv()
	IPAddr	= H_TO_NUDINT(TCPserv_1.ipaddr)
	Port	= TCPserv_1.portb
	NEWSTEP = 2
ENDIF

;Server to listening - until PC connects
IF STEP = 2 THEN
	TCPserv_1 FUB TCPserv()
	IPAddr	= H_TO_NUDINT(TCPserv_1.ipaddr)
	Port	= TCPserv_1.portb
	IF TCPserv_1.status = 0 THEN
		PLS = TRUE
		NEWSTEP = 3
	ELSE IF TCPserv_1.status = 27155 THEN 							;27155 = No buffer space available
		NEWSTEP = 6
	ENDIF
ENDIF

;PC Connected - if error then disconnect
IF STEP = 3 THEN

	WriteEnable = FALSE

	IF TCPsend_1.status = 0 THEN

		TCPrecv_1.enable = 1
		TCPrecv_1.cident = TCPserv_1.cident
		TCPrecv_1.buffer = ADR(rdata[0])
		TCPrecv_1.mxbuflng = SIZEOF(rdata)
		TCPrecv_1 FUB TCPrecv()
		RXLength = TCPrecv_1.rxbuflng
		RXStatus = TCPrecv_1.status

		IF RXLength > 0 THEN

			Data_RXTX_Type  = rdata[1] 								;WR = 1  WW = 3
			Data_Array_Type = rdata[2]								;C  = 1 D  = 2 Bag = 3

			Data_StartH = rdata[3]
			Data_Start 	= LSL(Data_StartH,8) + rdata[4]
			Data_AmountH = rdata[5]
			Data_Amount = LSL(Data_AmountH,8) + rdata[6]

			IF Data_Array_Type = 1 THEN
				Data_array_adr 	= pC
				Bytes			= 2
			ELSE IF Data_Array_Type = 2 THEN
				Data_array_adr = pD
				Bytes			= 2
			ELSE IF Data_Array_Type = 3 THEN
				Data_array_adr 	= pBag
				Bytes			= SIZEOF(Bag[0])
			ELSE IF Data_Array_Type = 4 THEN
;				Data_array_adr 	= pRB_Posn
;				Bytes			= SIZEOF(RB_Posn[0])
			ELSE IF Data_Array_Type = 5 THEN
				Data_array_adr 	= pD32
				Bytes			= SIZEOF(D32[0])
			ELSE IF Data_Array_Type = 6 THEN
;				Data_array_adr 	= pMCN
;				Bytes			= SIZEOF(MCN[0])
			ENDIF

			PacketID = rdata[RXLength - 1] ;Packet ID sent back to Driver for check

			;Increase tx_frame and rx frame now 5000 bytes (Data_Amount based on 16 bit register 2 bytes)
			Data_Valid = ((Data_RXTX_Type > 0) AND (Data_Array_Type > 0) AND (Data_array_adr > 0) AND (Data_Amount > 0) AND (Data_Amount <= 2500))

			IF Data_Valid THEN

				RXValid = RXValid + 1

				IF (Data_RXTX_Type = 1) THEN					;Word Read - Transmit Data to PC

					tx_frame[0] = rdata[0]						;PLC Station

					memcpy(adr(tx_frame[1]),Data_array_adr + (Data_Start * Bytes),(Data_Amount * Bytes))

					tx_frame[(Data_Amount * Bytes) + 1] = PacketID ;USINT(0) ;Checksum not required
					tx_length 	= (Data_Amount * Bytes) + 2
					WriteEnable = TRUE

				ELSE IF (Data_RXTX_Type = 3) THEN 				;Word Write - Receive data from PC

					LengthValid = (RXLength > (Data_Amount * Bytes))
					IF LengthValid THEN
						memcpy(Data_array_adr + (Data_Start * Bytes),adr(rdata[7]),(Data_Amount * Bytes))

						tx_frame[0] = $06							;ACK
						tx_frame[1] = rdata[0]						;PLC Station
						tx_length 	= 2
						WriteEnable	= TRUE							;Set write enable
					ELSE
						tx_frame[0] = $15 							;NAK
						tx_frame[1] = rdata[0] 						;PLC Station
						tx_length 	= 2
						WriteEnable	= TRUE							;Set write enable

					ENDIF

				ENDIF

			ELSE

				tx_frame[0] = $15 								;NAK
				tx_frame[1] = rdata[0] 							;PLC Station
				tx_length 	= 2
				WriteEnable	= TRUE								;Set write enable

			ENDIF

			IF WriteEnable THEN
				TCPsend_1.enable = 1
    			TCPsend_1.cident = TCPserv_1.cident
    			TCPsend_1.buffer = ADR(tx_frame[0])
    			TCPsend_1.buflng = tx_length ;SIZEOF(tx_frame)
    			TCPsend_1 FUB TCPsend()
	    	ENDIF

	    ENDIF

	ELSE
		TCPsend_1 FUB TCPsend()
	ENDIF

    IF (((TCPsend_1.status <> 0) AND (TCPsend_1.status <> 65535)) OR NoData) THEN
    	NoData  = FALSE
    	NEWSTEP = 4
    ENDIF

ENDIF
TON_10ms(((STEP = 3) AND (RXLength = 0)),500,NoData,NoDataET)

;Close the connection - if closed then go-to listen else go-to wait for close
IF STEP = 4 THEN
	TCPclose_1.enable = 1
	TCPclose_1.cident = TCPserv_1.cident
	TCPclose_1 FUB TCPclose()
	NEWSTEP = 5
ENDIF

;Closing - wait until connection closed
IF STEP = 5 THEN
	IF TCPclose_1.status <> 0 THEN
		TCPclose_1 FUB TCPclose()
	ELSE IF TCPclose_1.status = 0 THEN
		TCPsend_1.status = 0
		NEWSTEP = 1
	ENDIF
ENDIF

IF STEP = 6 THEN
	;Warm / Cold Start Required
ENDIF

;------------
;Connection 2
;------------

;Restart - from init routine
IF ResetConnection THEN
	IF EnableConnection2 THEN
		NEWSTEP2 = 1
	ELSE
		NEWSTEP2 = 0
	ENDIF
ENDIF

STEP2 = NEWSTEP2

;Disabled
IF STEP2 = 0 THEN
	;Do Nothing
ENDIF

;Init Server
IF STEP2 = 1 THEN
	TCPserv_2.enable = 1
	TCPserv_2.porta = 21002
	TCPserv_2 FUB TCPserv()
	IPAddr2	= H_TO_NUDINT(TCPserv_2.ipaddr)
	Port2	= TCPserv_2.portb
	NEWSTEP2 = 2
ENDIF

;Server to listening - until PC connects
IF STEP2 = 2 THEN
	TCPserv_2 FUB TCPserv()
	IPAddr2	= H_TO_NUDINT(TCPserv_2.ipaddr)
	Port2	= TCPserv_2.portb
	IF TCPserv_2.status = 0 THEN
		PLS2 = TRUE
		NEWSTEP2 = 3
	ELSE IF TCPserv_2.status = 27155 THEN								;27155 = No buffer space available
		NEWSTEP2 = 6
	ENDIF
ENDIF

;PC Connected - if error then disconnect
IF STEP2 = 3 THEN

	WriteEnable2 = FALSE

	IF TCPsend_2.status = 0 THEN

		TCPrecv_2.enable = 1
		TCPrecv_2.cident = TCPserv_2.cident
		TCPrecv_2.buffer = ADR(rdata2[0])
		TCPrecv_2.mxbuflng = SIZEOF(rdata2)
		TCPrecv_2 FUB TCPrecv()
		RXLength2 = TCPrecv_2.rxbuflng
		RXStatus2 = TCPrecv_2.status

		IF RXLength2 > 0 THEN

			Data_RXTX_Type  = rdata2[1] 								;WR = 1 BR = 2 WW = 3 BW = 4 - Bit Read and Bit Write not used
			Data_Array_Type = rdata2[2]									;C  = 1 D  = 2 E  = 3

			Data_StartH = rdata2[3]
			Data_Start 	= LSL(Data_StartH,8) + rdata2[4]
			Data_AmountH = rdata2[5]
			Data_Amount = LSL(Data_AmountH,8) + rdata2[6]

				IF Data_Array_Type = 1 THEN
				Data_array_adr 	= pC
				Bytes			= 2
		ELSE IF Data_Array_Type = 2 THEN
				Data_array_adr = pD
				Bytes			= 2
			ELSE IF Data_Array_Type = 3 THEN
				Data_array_adr 	= pBag
				Bytes			= SIZEOF(Bag[0])
			ELSE IF Data_Array_Type = 4 THEN
;				Data_array_adr 	= pRB_Posn
;				Bytes			= SIZEOF(RB_Posn[0])
			ELSE IF Data_Array_Type = 5 THEN
				Data_array_adr 	= pD32
				Bytes			= SIZEOF(D32[0])
			ELSE IF Data_Array_Type = 6 THEN
;				Data_array_adr 	= pMCN
;				Bytes			= SIZEOF(MCN[0])
			ENDIF

			PacketID = rdata2[RXLength2 - 1] ;Packet ID sent back to Driver for check

			Data_Valid = ((Data_RXTX_Type > 0) AND (Data_Array_Type > 0) AND (Data_array_adr > 0) AND (Data_Amount > 0) AND (Data_Amount < 1001))

			IF Data_Valid THEN

				RXValid2 = RXValid2 + 1

				IF (Data_RXTX_Type = 1) THEN							;Word Read - Transmit Data to PC

					tx_frame2[0] = rdata2[0] 							;PLC Station

					memcpy(adr(tx_frame2[1]),Data_array_adr + (Data_Start * Bytes),(Data_Amount * Bytes))

					tx_frame2[(Data_Amount * Bytes) + 1] = PacketID ;USINT(0) ;Checksum not required
					tx_length2 	= (Data_Amount * Bytes) + 2
					WriteEnable2 = TRUE

				ELSE IF (Data_RXTX_Type = 3) THEN 						;Word Write - Receive data from PC

					LengthValid = (RXLength2 > (Data_Amount * Bytes))
					IF LengthValid THEN
						memcpy(Data_array_adr + (Data_Start * Bytes),adr(rdata2[7]),(Data_Amount * Bytes))

						tx_frame2[0] = $06									;ACK
						tx_frame2[1] = rdata2[0] 							;PLC Station
						tx_length2 	= 2
						WriteEnable2	= TRUE								;Set write enable
					ELSE
						tx_frame2[0] = $15 									;NAK
						tx_frame2[1] = rdata2[0] 							;PLC Station
						tx_length2 	 = 2
						WriteEnable2 = TRUE									;Set write enable
					ENDIF
				ENDIF

			ELSE

				tx_frame2[0] = $15 										;NAK
				tx_frame2[1] = rdata2[0] 								;PLC Station
				tx_length2 	 = 2
				WriteEnable2 = TRUE										;Set write enable

			ENDIF

			IF WriteEnable2 THEN
				TCPsend_2.enable = 1
    			TCPsend_2.cident = TCPserv_2.cident
    			TCPsend_2.buffer = ADR(tx_frame2[0])
    			TCPsend_2.buflng = tx_length2 ;SIZEOF(tx_frame)
    			TCPsend_2 FUB TCPsend()
	    	ENDIF

	    ENDIF

	ELSE
		TCPsend_2 FUB TCPsend()
	ENDIF

    IF (((TCPsend_2.status <> 0) AND (TCPsend_2.status <> 65535)) OR NoData2) THEN
    	NoData2  = FALSE
    	NEWSTEP2 = 4
    ENDIF

ENDIF
TON_10ms(((STEP2 = 3) AND (RXLength2 = 0)),500,NoData2,NoData2ET)

;Close the connection - if closed then go-to listen else go-to wait for close
IF STEP2 = 4 THEN
	TCPclose_2.enable = 1
	TCPclose_2.cident = TCPserv_2.cident
	TCPclose_2 FUB TCPclose()
	NEWSTEP2 = 5
ENDIF

;Closing - wait until connection closed
IF STEP2 = 5 THEN
	IF TCPclose_2.status <> 0 THEN
		TCPclose_2 FUB TCPclose()
	ELSE IF TCPclose_2.status = 0 THEN
		TCPsend_2.status = 0
		NEWSTEP2 = 1
	ENDIF
ENDIF

IF STEP2 = 6 THEN
	;Warm / Cold Start Required
ENDIF

;Clear Reset Connection from Init Sub
ResetConnection = FALSE
END_PROGRAM
```

- Program Logical/Sequences/10ms/zzForceO (IEC) - * PLC Output forcing from graphics (no source held here)

### Program Logical/Sequences/10ms/zzIO (IEC) - * PLC Inputs and Outputs to Graphics

#### zzio.var
```iecst
VAR
	OutputCard : BIT_ENCODE;
	CurrentCard : UINT;
	InputCard : BIT_ENCODE;
	n : UINT;
	DataRegister : UINT;
END_VAR
```

- Program Logical/Sequences/10ms/zzOk (IEC) - * PLC Status to Graphics (no source held here)

### Package Logical/Sequences/200ms - 200ms Tasks

- Program Logical/Sequences/200ms/zzClearMem (IEC) - * Clear Permanent Memory (no source held here)

### Program Logical/Sequences/200ms/zzWeigh (IEC, version 6.00.0) - * Station Weight Calculation and Calibration

#### zzweigh.var
```iecst
VAR
	n : {REDUND_UNREPLICABLE} UINT;
	WeightUnits : {REDUND_UNREPLICABLE} DINT;
	StnHigh : {REDUND_UNREPLICABLE} UINT;
	StnLow : {REDUND_UNREPLICABLE} UINT;
	StnTestWgt : {REDUND_UNREPLICABLE} UINT;
	HighLow : {REDUND_UNREPLICABLE} UDINT;
	RawLow : {REDUND_UNREPLICABLE} DINT;
	StnRaw : {REDUND_UNREPLICABLE} ARRAY[0..99] OF UINT;
	NewLow : {REDUND_UNREPLICABLE} UINT;
	NewHigh : {REDUND_UNREPLICABLE} UINT;
	tstRaw : {REDUND_UNREPLICABLE} DINT;
	myRaw : {REDUND_UNREPLICABLE} DINT;
	myStnRaw : {REDUND_UNREPLICABLE} UINT;
	UseAI2744 : {REDUND_UNREPLICABLE} BOOL;
	FixCalibration : {REDUND_UNREPLICABLE} BOOL;
	Auto_ForceCalib : {REDUND_UNREPLICABLE} BOOL;
	Calib_Stn : {REDUND_UNREPLICABLE} UINT;
	Auto_Calib : {REDUND_UNREPLICABLE} enum_Calib;
END_VAR
```

#### zzweigh.ab
```automation-basic
PROGRAM _CYCLIC
	(* cyclic program *)

;---------------------------------------------------------------------------------------------
;Revision 1.00 01/05/2001 D.J. First Issu
;Revision 2.00 23/10/2002 D.J. WeightUnits changed to DINT (problem when raw values over 32767
;Revision 3.00 22/08/2006 D.J. Changed for AI261
;Revision 4.00 10/12/2009 D.J. Changed Calibration Storage Registers to D4400 etc.. AND AI2744
;Revision 5.00 09/08/2012 D.J. Changed Raw value to WeightRaw
;Revision 6.00 28/11/2012 D.J. Added Value Calibration values send to TrackView
;---------------------------------------------------------------------------------------------

;---------------------------------------------------------------------
;WeighStation Calibration and Weight Calculation - With AI261 & AI2744
;---------------------------------------------------------------------

UseAI2744 = TRUE ;Set PLC module type
IF Auto_ForceCalib THEN
	IF (Calib_Stn = 0) THEN
		Calib_Stn = 1
	ELSE IF Calib_Stn >= Std.MaxWeighstations THEN
		Calib_Stn = 0
		Auto_ForceCalib = FALSE
	ENDIF
	D[940 + Calib_Stn] = 1
	CASE Auto_Calib OF
		ACTION Calib_Low:
			D[995] = Calib_Stn
			D[996] = 11
			AI261Raw[Calib_Stn] = 0
			Auto_Calib = Calib_High
		ENDACTION

		ACTION Calib_High:
			D[995] = Calib_Stn
			D[996] = 12
			D[997] = 200
			AI261Raw[Calib_Stn] = 20000
			Auto_Calib = Calib_Low
			INC Calib_Stn
		ENDACTION
	ENDCASE
ENDIF

;divide by 1000 (AI261) or 100 (AI2744) should give around 50 parts per kg and keep raw value within UINT
;Add 32000 to value to ensure always positive
LOOP n = 1 TO (Std.MaxWeighstations + 20) DO
	;To view a particular stn then set tstRaw to the required stn

	IF tstRaw > 0 THEN
		myRaw = tstRaw ;AI261Raw[tstRaw]
	ELSE
		myRaw = ((AI261Raw[n] + AI261Raw[n + 30])/2)
	ENDIF
	;Ensure raw value is within + 24bit if out of range + 32bit
	IF (myRaw = $7FFFFFFF) THEN
		myRaw = $FFFFFF
	ENDIF
	;Ensure raw value is within - 24bit if out of range - 32bit
	IF (myRaw = $80000001) THEN
		myRaw = $FF000001
	ENDIF
	;Convert raw to UINT the 3 least significant digits are removed
	IF UseAI2744 THEN
		myStnRaw = UINT((myRaw / 100) + 32000)
	ELSE
		myStnRaw = UINT((myRaw / 1000) + 32000)
	ENDIF
	StnRaw[n] = myStnRaw
ENDLOOP

LOOP n = 1 TO Std.MaxWeighstations DO

	StnLow 		= D[4400 + n]
	StnHigh 	= D[4500 + n]
	StnTestWgt 	= D[4600 + n]

	;Calibrate Low - From TrackView
	IF (D[995] = n) AND (D[996] = 11) THEN
		NewLow = StnRaw[n]
		IF (NewLow > 0) AND (NewLow < $FFFF) THEN
			D[4400 + n] = NewLow
		ENDIF
		D[996] = 0 ;Cancel the Cal-Low
	ENDIF
	;Calibrate High - From TrackView
	IF (D[995] = n) AND (D[996] = 12) AND (D[997] > 0) THEN
		NewHigh = StnRaw[n]
		IF (NewHigh > 0) AND (NewHigh < $FFFF) AND (NewHigh > StnLow) THEN
			D[4500 + n] = NewHigh
			D[4600 + n] = D[997]		;Test-Weight
		ENDIF
		D[996] = 0 ;Cancel the Cal-High
	ENDIF

	;Weigh Calculation - Multiply up to give accurate results
	HighLow = StnHigh - StnLow
	HighLow = HighLow * 1000
	;Avoid "Divide By Zero"
	IF (StnTestWgt > 0) THEN
		WeightUnits = DINT(HighLow / StnTestWgt)
		RawLow = INT(StnRaw[n] - StnLow)
		RawLow = RawLow * 1000
		IF (WeightUnits > 0) THEN ;AND (RawLow > 0) THEN
			Stn[n].Weight = INT(RawLow / WeightUnits)
		ELSE
			Stn[n].Weight = 0
		ENDIF
	ELSE
		Stn[n].Weight = 999
	ENDIF

	;Calibration Values to TrackView when requested equals current station
	IF (D32[230] = n) THEN
		D32[231] = UDINT(n)
		D32[232] = UDINT(StnLow)
		D32[233] = UDINT(StnHigh)
		D32[234] = UDINT(StnTestWgt)
		D32[235] = UDINT(StnRaw[n])
		D32[236] = UDINT(Stn[n].Weight)
	ENDIF

ENDLOOP

END_PROGRAM
```

### Program Logical/Sequences/200ms/zzStn_Q (IEC, version 3.00.0) - * Stations into Q

#### zzstn_q.ab
```automation-basic
;Sorting Stations Into Q with provision for Pushbutton into Q
;------------------------------------------------------------

;Set "AutoMaticRelease" in "zzconst"
;Nothing to change!

;-------------------------------------------------------------------------------------
;Version 1.00 - 19/12/2005 D.J. First Issue
;Version 2.00 - 10/12/2009 D.J. Changed Setpoint Registers to D4000's
;Version 3.00 - 03/02/2011 D.J. Re-instated calibration stops release
;Version 4.00 - 13/09/2012 D.J. Allow for multiple station release with manual release
;-------------------------------------------------------------------------------------

PROGRAM _INIT
	LOOP n = 1 TO Std.MaxWeighstations DO
		Stn[n].ManRelease 	= 0
		D[800 + n]			= 0
	ENDLOOP
END_PROGRAM
PROGRAM _CYCLIC

StnsInQ 	= FALSE
StnsToPurge = FALSE

Calibration = (D[998] > 0)

LOOP z = 1 TO Std.MaxWeighstations DO

	n = z

	;Force to Single station for testing / monitoring
	IF TestStation > 0 THEN
		n = TestStation
	ENDIF

	ManualRelease 	= (D[800 + n] > 0)

	;For testing force valid weight values
	IF TestWeight > 0 THEN
		Stn[n].Weight = TestWeight
	ENDIF

	;If Current weight is less than the Min Release Weight or SP2 is set below the Min Release Weight or SP3 is set below the Min Release Weight
	ValidWeight = ((Stn[n].Weight > Std.MinReleaseWeight) AND (D[4800 + n] > Std.MinReleaseWeight) AND  (D[4900 + n] > Std.MinReleaseWeight))

	;Zurich Test - min release at 10kg
	;ValidWeight = ((Stn[n].Weight > 100) AND (D[4800 + n] > 100) AND  (D[4900 + n] > 100))

	;SP1 Reached - Approaching Weight
	SP1Reached = (Stn[n].Weight > D[4700 + n])

	;SP2 Reached - At Release Weight
	SP2Reached = (Stn[n].Weight > D[4800 + n])

	;SP3 Reached - Over Weight
	SP3Reached = (Stn[n].Weight > D[4900 + n])

	;Manual Release from TrackView
	IF ManualRelease THEN
		Stn[n].ManRelease 	= D[800 + n]
		D[800 + n] 			= 0 ;Cancel the Manual Release
	ENDIF

	IF PurgeStation THEN
		StnsToPurge = TRUE
	ENDIF

	;Enter Station into Q
	StnIntoQ = FALSE
	IF (Std.AutoMaticRelease AND SP2Reached AND ValidWeight AND (NOT SP3Reached)) THEN
		StnIntoQ = TRUE
	ELSE IF ((NOT Std.AutoMaticRelease) AND Stn[n].ReleaseButton AND SP2Reached AND ValidWeight AND (NOT SP3Reached)) THEN
		StnIntoQ = TRUE
	ELSE IF ((NOT Std.AutoMaticRelease) AND Stn[n].ReleaseButton AND Std.EnableOverUnderRelease AND ValidWeight) THEN
		StnIntoQ = TRUE
	ELSE IF (Stn[n].ManRelease = n) THEN
		StnIntoQ = TRUE ;Only put the Master for manual release into the Q
	ELSE IF ((D[7900 + n] > 1) AND Stn[n].CloseFlap AND ValidWeight) THEN
		StnIntoQ = TRUE ;Once loading flap has been closed then keep in Q
	ENDIF

	;Don't allow station release if calibrating
	IF Calibration THEN
		StnIntoQ = FALSE
	ENDIF

	IF StnIntoQ THEN
		StnsInQ = TRUE
		IF (Stn[n].QTime < $7FFF) THEN ;Keep within Integer range for PC
			Stn[n].QTime = (Stn[n].QTime + 1)
		ENDIF
	ELSE
		Stn[n].QTime = 0
	ENDIF

	D[100 + n] = Stn[n].QTime ;Set the time in the Q for Use by PC

	Stn[n].SP1	= FALSE
	Stn[n].SP2	= FALSE
	Stn[n].SP3	= FALSE

	IF SP3Reached THEN
		Stn[n].SP3 = TRUE
	ELSE IF SP2Reached OR StnIntoQ THEN
		Stn[n].SP2 = TRUE
	ELSE IF SP1Reached THEN
		Stn[n].SP1 = TRUE
	ENDIF

ENDLOOP

Std.StnsInQ 	= StnsInQ
Std.StnsToPurge = StnsToPurge

END_PROGRAM
```

### Program Logical/Sequences/200ms/zzAlarms (IEC) - Alarms - Messages and History

#### zzalarms.var
```iecst
VAR RETAIN
	I_CancelAlarm : BOOL;
END_VAR
VAR
	BuildD220 : UINT;
	AlmNumber : UINT;
	n : UINT;
	AlarmCount : UINT;
	CancelBeacon : BOOL;
	I_MotorOverload : BOOL;
	UnloadingAlarm : BOOL;
	I_InverterFault : BOOL;
	BeaconInList : BOOL;
	ConstKeep : UINT;
	I_SystemStopped : BOOL;
	AlarmOutput : ARRAY[0..9] OF BOOL;
	tmrAlmOutput : ARRAY[0..9] OF TON_10ms;
	I_SafetyHighLevel : BOOL;
	I_Safetyloading : BOOL;
	I_SafetyVC : ARRAY[0..2] OF BOOL;
	x : INT;
	AlarmZoneActive : ARRAY[0..99] OF BOOL;
	myZone : UINT;
END_VAR
```

#### zzalarms.ab
```automation-basic
PROGRAM _CYCLIC
	(* cyclic program *)

;-----------------------------------------------
;Alarm Messages with Screen position and history
;-----------------------------------------------

;-----------------------------------------------------------------
;Version 1.00 - 08/12/2005 First Issue D.J.
;Version 2.00 - 17/10/2006 Added Alarm.Extra D.J.
;Version 3.00 - 23/04/2007 Added Constants to stop them being lost
;Version 4.00 - 01/12/2009 Changed to 200 from 100 Sequence Alarms
;-----------------------------------------------------------------

;Alarm Constnts
ConstKeep = almBagDataError
ConstKeep = almBagNotArrived
ConstKeep = almBagNotAtProx
ConstKeep = almBagNotReleased
ConstKeep = almBagNotSettled
ConstKeep = almBagNotShownOnScreen
ConstKeep = almBagOverWeight
ConstKeep = almCarriageMoveFault
ConstKeep = almClearingBeltPleaseWait
ConstKeep = almDestinationNotValid
ConstKeep = almEmergencyStop
ConstKeep = almGeneralSequence
ConstKeep = almInverterFault
ConstKeep = almLoadNotDropped
ConstKeep = almMotorOverload
ConstKeep = almNoAlarm
ConstKeep = almPhotocellBlocked
ConstKeep = almPhotocellNotMade
ConstKeep = almStationNotClosed
ConstKeep = almStationNotEmpty
ConstKeep = almSwitchFault
ConstKeep = almUldNoBag
ConstKeep = almUldProgFinished
ConstKeep = almSystemStopped

;Note - Sequence must set the following
;Alarm[x].on
;Alarm[x].Bag - for the bag position where the alarm will appear
;Alarm[x].Name - for the message that will be displayed use constants strating "alm"
;Alarn[x].Extra - Extra data for Graphics to use ie. Line number with fault on offgoing storage

I_CancelAlarm 	= FALSE ;X[4].X16
I_EStop 		= Std.EStop; OR Std.EStopLoading
I_MotorOverload = Std.MotorOverload OR Std.MotorOverloadLoading
I_SystemStopped = NOT Std.SafetyOn
I_InverterFault = FALSE ;(X[3].X03 OR X[3].X04 OR X[3].X05 OR X[3].X06)
;I_SafetyHighLevel	= Std.HaltSysZone[myZone]
;I_Safetyloading		= Std.HaltSysLoading
;I_SafetyVC[1]		= Std.HaltSysVC[1]
;I_SafetyVC[2]		= Std.HaltSysVC[2]
;--------------
;Alarm Messages
;--------------

IF NOT Std.FireAlarm THEN
	Alarm[200].On	= TRUE
	Alarm[200].Bag 	= 0
	Alarm[200].Name	= ALM_FIREALARM;
ELSE IF I_EStop THEN
	Alarm[200].On	= TRUE
	Alarm[200].Bag 	= 0
	Alarm[200].Name	= almEmergencyStop
ELSE IF I_MotorOverload THEN
	Alarm[200].On	= TRUE
	Alarm[200].Bag 	= 0
	Alarm[200].Name	= almMotorOverload
ELSE IF I_SystemStopped THEN
	Alarm[200].On	= TRUE
	Alarm[200].Bag 	= 0
	Alarm[200].Name	= almSystemStopped
ELSE IF I_InverterFault THEN
	Alarm[200].On	= TRUE
	Alarm[200].Bag 	= 0
	Alarm[200].Name	= almInverterFault
ELSE
	Alarm[200].On	= FALSE
	Alarm[200].Bag 	= 0
	Alarm[200].Name	= almNoAlarm
ENDIF
LOOP n = 5 TO 9 DO
	Alarm[200 + n].On	= FALSE
	Alarm[200 + n].Bag 	= 0
	Alarm[200 + n].Name	= almNoAlarm
ENDLOOP
IF I_SafetyHighLevel THEN
	Alarm[205].On	= TRUE
	Alarm[205].Bag 	= 0
	Alarm[205].Name	= almSafetyHighLevel
ENDIF
IF I_Safetyloading THEN
	Alarm[206].On	= TRUE
	Alarm[206].Bag 	= 0
	Alarm[206].Name	= almSafetyLoading
ENDIF
IF I_SafetyVC[1] THEN	 ; Don't use VC alarms unless cust reqs as will
	Alarm[207].On	= TRUE
	Alarm[207].Bag 	= 0
	Alarm[207].Name	= almSafetyVC
	Alarm[207].Extra = 1
ENDIF
;IF I_SafetyVC[2] THEN
;	Alarm[208].On	= TRUE
;	Alarm[208].Bag 	= 0
;	Alarm[208].Name	= almSafetyVC
;	Alarm[208].Extra = 2
;ENDIF
;

;Shuffle the Alarms List

AlarmCount 		= 0
BeaconInList 	= FALSE
LOOP x = 0 TO Std.MaxZones DO
	AlarmZoneActive[x] = FALSE
ENDLOOP

LOOP n = 1 TO 10 DO

	;If Alarm not on anymore the clear from the list
	AlmNumber = D[200 + n]
	IF NOT Alarm[AlmNumber].On THEN
		D[200 + n] = 0
		D[210 + n] = 0
	ENDIF

	;Shuffle the list down
	IF (D[200 + n] = 0) AND (D[201 + n] > 0) AND (n <> 10) THEN
		D[200 + n] = D[201 + n]
		D[210 + n] = D[211 + n]
		D[201 + n] = 0
		D[211 + n] = 0
	ENDIF

	;Set InList for any alarm in the list
	Alarm[D[200 + n]].InList = TRUE

	;Calculate total alarms in the list
	IF D[200 + n] > 0 THEN
		AlarmCount = AlarmCount + 1
	ENDIF
	myZone = Alarm[D[200 + n]].Zone
	;Is the alarm beacon required?
	IF Alarm[AlmNumber].On AND Alarm[AlmNumber].Beacon THEN
		BeaconInList = TRUE
		IF (myZone <= Std.MaxZones) AND Alarm[D[200 + n]].InList  THEN
			AlarmZoneActive[myZone] = TRUE
		ENDIF
	ENDIF

ENDLOOP

;Cancel the alarm beacon
IF I_CancelAlarm THEN
	CancelBeacon = TRUE
ENDIF

;Cancel the CancelAlarm beacon if no alarm in the list requires the beacon
IF NOT BeaconInList THEN
	CancelBeacon = FALSE
ENDIF

;Look at each sequence alarm and if not in list then add to list if space
LOOP n = 1 TO 209 DO

	;If alarm active and a code has been given and not in the list and history is clear then add
	IF ((AlarmCount < 10) AND Alarm[n].On AND NOT Alarm[n].InList AND ((D[221] = 0) OR (n > 200))) THEN

		;If name not set then set to general
		IF (Alarm[n].Name = 0) THEN
			Alarm[n].Name = almGeneralSequence
		ENDIF

		D[210] 			= n
		BuildD220		= LSL(Alarm[n].Extra,8)
		BuildD220 		= BuildD220 + Alarm[n].Name
		D[220] 			= BuildD220

		;New alarm found requiring the beacon
		IF Alarm[n].Beacon THEN
			CancelBeacon = FALSE
		ENDIF

		;Store to History - if not Unloading Alarm
		IF (n <= 200) THEN
			D[221] 			= n				;Alarm Number (Seq)
			D[222]			= Alarm[n].Name	;Alarm Name / Message
			D[223] 			= D[223] + 1	;Alarm ID
			D[224]			= Alarm[n].Extra;Alarm Extra Data
			IF D[223] > 32000 THEN
				D[223] = 1
			ENDIF
		ENDIF

		;Inc Total Alarms
		AlarmCount = AlarmCount + 1

	ENDIF

	;Cancel All InList's - will be checked on the next scan
	Alarm[n].InList = FALSE

ENDLOOP

;Show Alarm position on the screen
IF D[201] > 0 THEN
	D[0] = Alarm[D[201]].Bag
ELSE
	D[0] = 0
ENDIF
;Alarms 203> used for extra safety zones
UnloadingAlarm = (Alarm[201].On OR Alarm[202].On OR Alarm[203].On OR Alarm[204].On OR Alarm[205].On OR Alarm[206].On); OR Alarm[207].On OR Alarm[208].On)

;Alarm Output - Unloading Alarm cannot be cancelled
;Y[3].Y01 = ((BeaconInList AND NOT CancelBeacon) OR UnloadingAlarm)
;Y[4].Y15 = CancelAlarm

;Timed Alarm Output Horn or Beacon

LOOP n = 0 TO Std.MaxZones DO
	AlarmOutput[n] = AlarmZoneActive[n] AND (BeaconInList OR UnloadingAlarm)
	tmrAlmOutput[n].IN = AlarmZoneActive[n] AND (BeaconInList OR UnloadingAlarm)
	tmrAlmOutput[n].PT = 3000
	tmrAlmOutput[n] FUB TON_10ms()

	AlarmOutput[n] = (AlarmZoneActive[n] AND (BeaconInList OR UnloadingAlarm) AND NOT tmrAlmOutput[n].Q)
ENDLOOP

	;Alarm for Panel 1

Y[1].Y01 = (AlarmOutput[0] OR AlarmOutput[1] OR AlarmOutput[2])
//Y[20].Y01 = (AlarmOutput[0] OR AlarmOutput[3] OR AlarmOutput[4])

END_PROGRAM
```

- Program Logical/Sequences/200ms/zzTime (IEC) - * System running time (no source held here)

### Program Logical/Sequences/200ms/USB_Pmem (IEC) - * USB - Backup and Restore data

#### usb_pmem.var
```iecst
VAR
	bOK	:BOOL;
	byErrorLevel	:USINT;
	CurrentFile	:UINT;
	STEP	:UINT;
	FOpen	:FileOpen;
	wStatus	:UINT;
	dwIdent	:UDINT;
	wError	:UINT;
	FCreate	:FileCreate;
	FWrite	:FileWrite;
	FRead	:FileRead;
	FClose	:FileClose;
END_VAR
```

### Package Logical/Sequences/200ms/udp_CTT - Sorting Station Displays

### Program Logical/Sequences/200ms/udp_CTT/UDP_CTT (IEC)

#### udp.var
```iecst
(********************************************************************
 * COPYRIGHT --
 ********************************************************************
 * Program: udp
 * File: udp.var
 * Author: flender
 * Created: November 05, 2009
 ********************************************************************
 * Local variables of program udp
 ********************************************************************)
VAR
	send_buffer : ARRAY[0..3] OF buffer_UDP_CTT;
	Remainder_a : UINT;
END_VAR
VAR RETAIN
	Start : BOOL;
	Start2 : BOOL;
END_VAR
VAR CONSTANT
	udpConnectionOk : USINT := 1;
END_VAR
VAR RETAIN
	UDPopen_1 : UDPopen;
	UDPsend_1 : UDPsend;
END_VAR
VAR
	Daten_senden : BOOL;
	pBaga : STRING[11];
	pBagb : STRING[11];
	pBagc : STRING[11];
	pBagd : STRING[11];
	pBaga_w : STRING[11];
	pBagb_w : STRING[11];
	pBagc_w : STRING[11];
	pBagd_w : STRING[11];
	unit : STRING[2];
	Maximum_PCTs : USINT;
	stat_index : UINT;
	buff_index : UINT;
	Maximum_CTTs : USINT;
	RX : BOOL;
	UDPrecv_1 : UDPrecv;
	IP_Adress_client : UDINT;
	bufferRX : RX_Buffer_CCT_PLC;
	show_long_id : BOOL;
	Remainder_b : UINT;
	WgtRound_a : UINT;
	WgtRound_b : UINT;
	Remainder_c : UINT;
	WgtRound_c : UINT;
	Remainder_d : UINT;
	WgtRound_d : UINT;
END_VAR
```

#### udp.ab
```automation-basic
PROGRAM _INIT

Start 	= TRUE		  ;enables the UDP Connection
Start2 	= TRUE
RX = TRUE

strcpy(adr(unit),"kg")	 ;The Unit of weight for the CTT
show_long_id = 1;	 Please change value to 1 to send long ID instead of Cat number

;-----------------------------------------------------
;ONLY FOR INFORMATION:
;-----------------------------------------------------
;D[5000] to D[5014] Customer Bank 1 upto 30 chr max.
;D[5020] to D[5034] Customer Bank 2 upto 30 chr max.
;D[5040] to D[5054] Customer Bank 3 upto 30 chr max.
;D[5060] to D[5074] Customer Bank 4 upto 30 chr max.
;D[5080] to D[5094] Customer Bank 5 upto 30 chr max.

;D[5100] to D[5114] Category Stn 1 Category Name 30 chr max
;D[5115] to D[5119] Long ID Stn 1 Max 10 chrs.

;D[5120] to D[5134] Category Stn 2 Category Name 30 chr max
;D[5135] to D[5139] Long ID Stn 2 Max 10 chrs.

;D[5140] to D[5154] Category Stn 3 Category Name 30 chr max
;D[5155] to D[5159] Long ID Stn 3 Max 10 chrs.

;...
;...
;-----------------------------------------------------

END_PROGRAM

(********************************************************************
 * COPYRIGHT --
 ********************************************************************
 * Program: udp
 * File: udp.ab
 * Author: flender
 * Created: November 05, 2009
 ********************************************************************
 * Implementation of program udp
 ********************************************************************)

PROGRAM _CYCLIC

;-----------------------------------------------------
; Open the UDP Connection
;-----------------------------------------------------

	if Start OR (UDPopen_1.status <> 0) THEN
		UDPopen_1.enable = 1
		UDPopen_1.port = 21003
		UDPopen_1 FUB UDPopen()
		Start = FALSE

;-----------------------------------------------------
; receive UDP Telegramm
;-----------------------------------------------------

	else if	 (RX AND (UDPopen_1.status = 0)) THEN
		UDPrecv_1.enable = 1
		UDPrecv_1.cident = UDPopen_1.cident
		UDPrecv_1.buffer = ADR(bufferRX)
		UDPrecv_1.buflng = SIZEOF(bufferRX)
		UDPrecv_1 FUB UDPrecv()
		if (bufferRX.sendRequest = 1)then
			bufferRX.sendRequest = 0
			RX = FALSE
		else
			RX = TRUE
		endif

;-----------------------------------------------------
; send UDP Telegramm
;-----------------------------------------------------

	else if(NOT RX and (UDPopen_1.status=0)) then

		Daten_senden = 0

		;-----------------------------------------------------
		;if connection is OK, the CTT needs this value for showing
		;-----------------------------------------------------
		send_buffer[0].UDP_OK = udpConnectionOk

		;-----------------------------------------------------
		;set up the customer name to sending buffer
		;-----------------------------------------------------
		;Customer Name for Station 1-12
		if (bufferRX.DwnLeft <= 12) then
			loop stat_index = 0 to 14 do
				send_buffer[0].Customer[stat_index] = (D[5000 + stat_index]) (* initialize the buffer *)
			endloop
		;Customer Name for Station 13-24
		else if (bufferRX.DwnLeft > 12) and (bufferRX.DwnLeft <= 24) then
			loop stat_index = 0 to 14 do
				send_buffer[0].Customer[stat_index] = (D[5020 + stat_index]) (* initialize the buffer *)
			endloop
		;Customer Name for Station 25-36
		else if (bufferRX.DwnLeft > 24) and (bufferRX.DwnLeft <= 36) then
			loop stat_index = 0 to 14 do
				send_buffer[0].Customer[stat_index] = (D[5040 + stat_index]) (* initialize the buffer *)
			endloop
		;Customer Name for Station 37-48
		else if (bufferRX.DwnLeft > 36) and (bufferRX.DwnLeft <= 48) then
			loop stat_index = 0 to 14 do
				send_buffer[0].Customer[stat_index] = (D[5060 + stat_index]) (* initialize the buffer *)
			endloop
		;Customer Name for Station 49-56
		else
			loop stat_index = 0 to 14 do
				send_buffer[0].Customer[stat_index] = (D[5080 + stat_index]) (* initialize the buffer *)
			endloop
		endif

		;-----------------------------------------------------
		;set the IP-Adress of the receiving CTT
		;-----------------------------------------------------
		UDPsend_1.ipaddr = 	UDPrecv_1.ipaddr

		;-----------------------------------------------------
		; Copy Category data to sending buffer
		;-----------------------------------------------------
		loop buff_index = 0 to 14 do
			send_buffer[0].Category[buff_index] = D[5100 + buff_index + (bufferRX.UpLeft-1)*20]
			send_buffer[1].Category[buff_index]	= D[5100 + buff_index + (bufferRX.DwnLeft-1)*20]
			send_buffer[2].Category[buff_index]	= D[5100 + buff_index + (bufferRX.UpRight-1)*20]
			send_buffer[3].Category[buff_index]	= D[5100 + buff_index + (bufferRX.DwnRight-1)*20]
		endloop

		if show_long_id = 0 then
			send_buffer[0].use_long_id = 0
			;-----------------------------------------------------
			; Copy Cat data to sending buffer
			;-----------------------------------------------------
			;Make a String of Bag.Cat
			udiToString(adr(pBaga),(Bag[200 + bufferRX.UpLeft].Cat),10)
			udiToString(adr(pBagb),(Bag[200 + bufferRX.DwnLeft].Cat),10)
			udiToString(adr(pBagc),(Bag[200 + bufferRX.UpRight].Cat),10)
			udiToString(adr(pBagd),(Bag[200 + bufferRX.DwnRight].Cat),10)
			;copy the string(10Byte)to sending buffer
			memcpy(adr(send_buffer[0].Cat[0]),adr(pBaga),10)
			memcpy(adr(send_buffer[1].Cat[0]),adr(pBagb),10)
			memcpy(adr(send_buffer[2].Cat[0]),adr(pBagc),10)
			memcpy(adr(send_buffer[3].Cat[0]),adr(pBagd),10)
		else
			send_buffer[0].use_long_id = 1
			;-----------------------------------------------------
			; Copy Long ID data to sending buffer
			;-----------------------------------------------------
			loop buff_index = 0 to 4 do
				send_buffer[0].Cat[buff_index] = D[5115 + buff_index + (bufferRX.UpLeft-1)*20]
				send_buffer[1].Cat[buff_index] = D[5115 + buff_index + (bufferRX.DwnLeft-1)*20]
				send_buffer[2].Cat[buff_index] = D[5115 + buff_index + (bufferRX.UpRight-1)*20]
				send_buffer[3].Cat[buff_index] = D[5115 + buff_index + (bufferRX.DwnRight-1)*20]
			endloop
		endif
		;-----------------------------------------------------
		; Copy Wgt data to sending buffer
		;-----------------------------------------------------

		;round up weight to give to CTT
		Remainder_a = SINT(Bag[200 + bufferRX.UpLeft].Wgt MOD 10)
		IF (Remainder_a > 4) THEN
			WgtRound_a = (Bag[200 + bufferRX.UpLeft].Wgt + 10)
		ELSE
			WgtRound_a = Bag[200 + bufferRX.UpLeft].Wgt
		ENDIF

		Remainder_b = SINT(Bag[200 + bufferRX.DwnLeft].Wgt MOD 10)
		IF (Remainder_b > 4) THEN
			WgtRound_b = (Bag[200 + bufferRX.DwnLeft].Wgt + 10)
		ELSE
			WgtRound_b = Bag[200 + bufferRX.DwnLeft].Wgt
		ENDIF

		Remainder_c = SINT(Bag[200 + bufferRX.UpRight].Wgt MOD 10)
		IF (Remainder_c > 4) THEN
			WgtRound_c = (Bag[200 + bufferRX.UpRight].Wgt + 10)
		ELSE
			WgtRound_c = Bag[200 + bufferRX.UpRight].Wgt
		ENDIF

		Remainder_d = SINT(Bag[200 + bufferRX.DwnRight].Wgt MOD 10)
		IF (Remainder_d > 4) THEN
			WgtRound_d = (Bag[200 + bufferRX.DwnRight].Wgt + 10)
		ELSE
			WgtRound_d = Bag[200 + bufferRX.DwnRight].Wgt
		ENDIF

		;Make a String of WgtRound
		udiToString(adr(pBaga_w),(WgtRound_a/10),3)
		udiToString(adr(pBagb_w),(WgtRound_b/10),3)
		udiToString(adr(pBagc_w),(WgtRound_c/10),3)
		udiToString(adr(pBagd_w),(WgtRound_d/10),3)
		;copy the string(3Byte)to sending buffer
		memcpy(adr(send_buffer[0].Wgt[0]),adr(pBaga_w),3)
		memcpy(adr(send_buffer[1].Wgt[0]),adr(pBagb_w),3)
		memcpy(adr(send_buffer[2].Wgt[0]),adr(pBagc_w),3)
		memcpy(adr(send_buffer[3].Wgt[0]),adr(pBagd_w),3)
		;copy the unit of weight (kg) to buffer
		memcpy(adr(send_buffer[0].Wgt[3]),adr(unit),2)
		memcpy(adr(send_buffer[1].Wgt[3]),adr(unit),2)
		memcpy(adr(send_buffer[2].Wgt[3]),adr(unit),2)
		memcpy(adr(send_buffer[3].Wgt[3]),adr(unit),2)

		;-----------------------------------------------------
		;set up the color for the background (at the moment a constant value)
		;-----------------------------------------------------
	    send_buffer[0].BackColor = 60
	    send_buffer[1].BackColor = 60
	    send_buffer[2].BackColor = 60
	    send_buffer[3].BackColor = 60

		;-----------------------------------------------------
		;make UDP port ready for sending data
		;-----------------------------------------------------
		UDPsend_1.enable = 1                		; enables the FBK
	   	UDPsend_1.cident = UDPopen_1.cident         ; copy the Ident number
		UDPsend_1.buffer = ADR(send_buffer)      	; address of the buffer
		UDPsend_1.buflng = SIZEOF(send_buffer)      ; size of the buffer
		UDPsend_1.port = 21000              		; port number of the receiver

		;-----------------------------------------------------
		;starts the sending process
		;-----------------------------------------------------

		UDPsend_1 FUB UDPsend()
		RX = TRUE
	endif

	;-----------------------------------------------------
	;starts the sending process when UDP Buisy
	;-----------------------------------------------------
	if (UDPsend_1.status = 65535) then
		UDPsend_1 FUB UDPsend()
	endif

END_PROGRAM
```

- Program Logical/Sequences/zzstnmix (IEC, version 1.00.0) - * Station mixing Customer and Categories (no source held here)

### Program Logical/Sequences/zzstatus (IEC, version 1.00.0) - * System status for edit bags

#### zzstatus.var
```iecst
VAR
	OngoingStopped	:BOOL;
	OffgoingStopped	:BOOL;
	LoadingStopped	:BOOL;
	tmrForce	:TON_10ms;
	ForceEnable	:BOOL;
END_VAR
```

### Program Logical/Sequences/zzstnser (IEC, version 1.00.0) - * Station Release Search

#### zzstnser.var
```iecst
VAR RETAIN
	SearchFound	:UINT;
	n	:UINT;
	LineSearchManual	:UINT;
	SearchLine	:UINT;
END_VAR

VAR
	Bank	:UINT;
	LineSearch	:ARRAY [0..4] OF UINT;
	Choice	:UINT;
END_VAR
```

#### zzstnserCyclic.ab
```automation-basic
PROGRAM _CYCLIC
	(* cyclic program *)

;Sorting Station Search Routine - No changes required!
;-----------------------------------------
;Revision 1.00 19/12/2005 First Issue D.J.
;-----------------------------------------

;Only one Bank / Loading VC can search in a given scan.

Bank = Bank + 1
IF (Bank > Std.MaxSearch) THEN
	Bank = 1
ENDIF

;Used by other sequences that need to check for Line[x].SpaceBIT direct
;eg. Loading VC will look for Enable.Search = 3
Enable.Search = Bank

IF (Bank <= Std.MaxStationBanks) THEN

	IF (Ldg[Bank].Search = 1) THEN

		Ldg[Bank].Found = 0
		Ldg[Bank].Line  = 0

		SearchFound = 0
		SearchLine  = 0

		Stn[0].QTime = 0

		LOOP n = Ldg[Bank].StartStn TO Ldg[Bank].EndStn DO

			IF ((Stn[n].QTime > 10) AND (Stn[n].QTime > Stn[0].QTime)) THEN

				;Destination has been given to bag by operator check
				LineSearchManual = Stn[n].DestManual

				;1st 2nd 3rd and 4th Line choices
				LineSearch[1]   = D[3000 + n]
				LineSearch[2]   = D[3100 + n]
				LineSearch[3]   = D[3200 + n]
				LineSearch[4]   = D[3300 + n]

				;Always Search for at least 1 space
				IF (Stn[n].SpacesRequired = 0) THEN
					Stn[n].SpacesRequired = 1
				ENDIF

				;When manual is selected then the 1st 2nd 3rd and 4th are not checked
				IF (LineSearchManual > 0) THEN
					IF (Line[LineSearchManual].SpaceBIT > 0) THEN
						SearchFound  		= n
						SearchLine   		= LineSearchManual
						Stn[0].QTime 		= Stn[n].QTime
						Ldg[Bank].Search   	= 2
					ENDIF
				ELSE
					;Check line choice 1st to 4th in order if any valid then exit loop
					LOOP Choice = 1 TO 4 DO
						IF (LineSearch[Choice] > 0) AND (Line[LineSearch[Choice]].SpaceBIT >= Stn[n].SpacesRequired) THEN
							SearchFound  		= n
							SearchLine   		= LineSearch[Choice]
							Stn[0].QTime 		= Stn[n].QTime
							Ldg[Bank].Search   	= 2

						ENDIF
						EXITIF (SearchFound > 0)
					ENDLOOP

				ENDIF

			ENDIF

		ENDLOOP

		IF (Ldg[Bank].Search = 2) THEN
			Ldg[Bank].Found  = SearchFound
			Ldg[Bank].Line   = SearchLine
		ELSE
			Ldg[Bank].Search = 0 ;Failed
		ENDIF

	ENDIF
ENDIF
END_PROGRAM
```

- Program Logical/Sequences/zztc2str (IEC, version 1.00.0) - * TC2 Start - Scan Time Calculation (no source held here)

### Program Logical/Sequences/zzstd (IEC) - * Standard Functions

#### zzstd.var
```iecst
VAR
	TimerClkB	:ARRAY [0..4] OF TON_10ms;
	TimerClkA	:ARRAY [0..4] OF TON_10ms;
	n	:UINT;
	TimerClkPT	:ARRAY [0..4] OF UINT;
END_VAR
```

#### zzstdCyclic.ab
```automation-basic
PROGRAM _CYCLIC
	(* cyclic program *)

;Version 1.00 First Issue
;Version 2.00 Added Bag[0] and Removed Mitsubishi M90xx's clock's

;Set all of bag 0 to Zero for use when deleting bags
Bag[0].Cat = 0
Bag[0].Dst = 0
Bag[0].Wgt = 0
Bag[0].Cnt = 0
Bag[0].Cus = 0
Bag[0].Day = 0
Bag[0].Spare = 0

;Standard Clocks
TimerClkPT[0] = 5 	;100ms
TimerClkPT[1] = 10 	;200ms
TimerClkPT[2] = 25 	;500ms
TimerClkPT[3] = 50 	;1s
TimerClkPT[4] = 100 ;2s

LOOP n = 0 TO 4 DO

	TimerClkA[n].IN = NOT TimerClkB[n].Q
	TimerClkA[n].PT = TimerClkPT[n]
	TimerClkA[n] FUB TON_10ms()

	TimerClkB[n].IN = TimerClkA[n].Q
	TimerClkB[n].PT = TimerClkPT[n]
	TimerClkB[n] FUB TON_10ms()

ENDLOOP

Std.Clock100ms 	= TimerClkA[0].Q
Std.Clock200ms 	= TimerClkA[1].Q ;M9031
Std.Clock500ms 	= TimerClkA[2].Q
Std.Clock1s 	= TimerClkA[3].Q ;M9032
Std.Clock2s 	= TimerClkA[4].Q ;M9033

Y[6].Y16 = NOT OK[1]
Y[7].Y13 = NOT OK[2]
Y[7].Y14 = NOT OK[3]
Y[7].Y16 = NOT OK[4]

Y[7].Y15 =  NOT OK[5]
END_PROGRAM
```

#### zzstdInit.ab
```automation-basic
PROGRAM _INIT
	(* init program *)

;Memory Address Pointers

;Note - pC was mem_adr_C in old programs
pC			= ADR(C)
pD			= ADR(D)
pBag		= ADR(Bag)

Zero 		= 0
END_PROGRAM
```

- Program Logical/Sequences/zzforcei (IEC, version 1.00.0) - * PLC Input forcing from fraphics (no source held here)

### Program Logical/Sequences/zzconst (IEC) - * System Constants - Adjust to Suit

#### zzconstInit.ab
```automation-basic
PROGRAM _INIT
	(* init program *)

Std.AutoMaticRelease   	= TRUE	;Set to TRUE for AutoMatic Release using setpoints. FALSE for Push-Button Release
Std.StationReports  	= TRUE  ;Transfer reports to PC

Std.PairingLoop   		= FALSE
Std.CustomerFIFO		= TRUE	;Use Customer FIFO Table

Std.MaxIO				= 39	;Max PLC I/O Cards - check X and Y array size

Std.MaxCats           	= 99	;Max Categories - Should be 99 or less Max = 255
Std.MaxCust           	= 999	;Max Customers
Std.MaxDischargers    	= 2		;Total Dischargers
Std.MaxLines          	= 11	    ;Max storage lines
Std.MaxLinesBuffers   	= 13	;Storage lines + Buffers
Std.MaxWeighstations  	= 16	    ;Total Weighstations
Std.MaxStationBanks		= 1		;Total Banks of sorting Stations
Std.MaxSearch			= 2    	;Include all station banks and Loading VC's etc
Std.StationBagsStart[1]	= 201	;Bag Number of first bank of sorting stations
Std.StationBagsStart[2] = 0 	;Bag Number of second bank of sorting stations
Std.MinReleaseWeight  	= 30	;Include 10ths Norm 30
Std.MaxKanLink               = 2

Ldg[1].StartStn 		= 1 	;Bank 1 Start station number
Ldg[1].EndStn			= 16	    ;Bank 1 End station number

Ldg[2].StartStn 		= 0 	;Bank 2 Start station number
Ldg[2].EndStn			= 0		;Bank 2 End station number

;Enter the First and Last bag for all the Storage lines including buffers
Line[1].FirstBag = 1
Line[1].LastBag  = 15

Line[2].FirstBag = 16
Line[2].LastBag  = 30

Line[3].FirstBag = 31
Line[3].LastBag  = 45

Line[4].FirstBag = 46
Line[4].LastBag  = 60

Line[5].FirstBag = 61
Line[5].LastBag  = 75

Line[6].FirstBag = 76
Line[6].LastBag  = 90

Line[7].FirstBag = 91
Line[7].LastBag  = 105

Line[8].FirstBag = 106
Line[8].LastBag  = 120

Line[9].FirstBag = 121
Line[9].LastBag  = 135

Line[10].FirstBag = 136
Line[10].LastBag  = 150

Line[11].FirstBag = 151
Line[11].LastBag  = 165

Line[12].FirstBag = 227
Line[12].LastBag  = 227

Line[13].FirstBag = 229
Line[13].LastBag  = 230

Line[14].FirstBag = 0
Line[14].LastBag  = 0

Line[15].FirstBag = 0
Line[15].LastBag  = 0

Line[16].FirstBag = 0
Line[16].LastBag  = 0

Line[17].FirstBag = 0
Line[17].LastBag  = 0

Line[18].FirstBag = 0
Line[18].LastBag  = 0

Line[19].FirstBag = 0
Line[19].LastBag  = 0

Line[20].FirstBag = 0
Line[20].LastBag  = 0

Line[21].FirstBag = 227
Line[21].LastBag  = 227

Line[22].FirstBag = 229
Line[22].LastBag  = 230

Line[23].FirstBag = 0
Line[23].LastBag  = 0

Line[24].FirstBag = 0
Line[24].LastBag  = 0

Line[25].FirstBag = 0
Line[25].LastBag  = 0

Line[26].FirstBag = 0
Line[26].LastBag  = 0

Line[27].FirstBag = 0
Line[27].LastBag  = 0

Line[28].FirstBag = 0
Line[28].LastBag  = 0

Line[29].FirstBag = 0
Line[29].LastBag  = 0

Line[30].FirstBag = 0
Line[30].LastBag  = 0

Line[31].FirstBag = 0
Line[31].LastBag  = 0

Line[32].FirstBag = 0
Line[32].LastBag  = 0

Line[33].FirstBag = 0
Line[33].LastBag  = 0

Line[34].FirstBag = 0
Line[34].LastBag  = 0
END_PROGRAM
```

### Program Logical/Sequences/zztrip (IEC) - * Counting Trips with debounce

#### zztrip.var
```iecst
VAR
	CountOld	:ARRAY [0..49] OF UINT;
	TripPLS	:ARRAY [0..49] OF R_TRIG;
	Timer	:ARRAY [0..49] OF TON_10ms;
	CountTrip	:ARRAY [0..49] OF BOOL;
	n	:UINT;
END_VAR
```

#### zztripCyclic.ab
```automation-basic
PROGRAM _CYCLIC
(* cyclic program *)

;--------------------------------------------------------------------------
;Primary trolley counting trips - ensure the main program can see the input
;--------------------------------------------------------------------------

CountTrip[1]  = X[4].X01 ;Bag on line 1
CountTrip[2]  = X[4].X02 ;            2
CountTrip[3]  = X[4].X03 ;            3
CountTrip[4]  = X[4].X04 ;            4
CountTrip[5]  = X[4].X05 ;Bag out sdc1
CountTrip[6]  = X[4].X06 ;            6
CountTrip[7]  = X[4].X07 ;            7
CountTrip[8]  = X[4].X08 ;            8
CountTrip[9]  = X[4].X09 ;            9
CountTrip[10] = X[4].X10 ;           10
CountTrip[11] = X[4].X11 ;           11
CountTrip[12] = X[3].X03 ;           12
CountTrip[13] = X[3].X07 ;           13
;CountTrip[14] = X[4].X14 ;           14
CountTrip[15] = X[5].X09
CountTrip[16] = X[5].X16 ;SVC1 Buffer full
;CountTrip[17] = X[4].X01 ;Bag on buffer line A
;CountTrip[18] = X[6].X13 ;Bag out of svc2
;CountTrip[19] = X[7].X03 ;Sdc4 Bag Out
;CountTrip[20] = X[6].X12 ;Sdc3 Bag Out
;CountTrip[21] = X[6].X16 ;Sdc1 buffer line full
;CountTrip[22] = X[6].X15 ;Sdc2 buffer line full
;CountTrip[23] = X[9].X16 ;Sdc3 buffer line full
;CountTrip[24] = X[9].X14 ;Sdc4 buffer line full
;CountTrip[25] = X[9].X12 ;Sdc5 buffer line full
;CountTrip[26] = X[7].X07 ;Sdc5 Bag Out
;CountTrip[27] = X[6].X05 ;Bag out of sdc1
;CountTrip[28] = X[6].X08 ;Bag out of sdc2
;CountTrip[29] = X[7].X08 ;Sbc1 Buffer line full
;CountTrip[30] = X[3].X11 ;Sic1 buffer line full
;CountTrip[31] = X[7].X13 ;Bag out of svc3
;CountTrip[32] = X[10].X06 ;Bag out offgoing bag stacker
;CountTrip[33] = X[8].X06 ; Bag out of loading unit
;CountTrip[34] = X[4].X16
;CountTrip[35] = X[7].X16 ;Sbc1 Bag out
;CountTrip[36] = X[3].X12 ;Bag on transit line B

LOOP n = 1 TO 22 DO

	TripPLS[n].CLK = CountTrip[n]
	TripPLS[n] FUB R_TRIG()

	IF TripPLS[n].Q AND Timer[n].Q AND (C[n] < 2) THEN
		C[n] = C[n] + 1
	ENDIF

	Timer[n].IN = NOT CountTrip[n]
	Timer[n].PT = 10 ;100 = 1second
	Timer[n] FUB TON_10ms()

	Line[n].Full 	= (C[n] = 1)
	Line[n].Clear 	= ((C[n] >= 2) AND Timer[n].Q)

	Line[n].Trip	= (((CountOld[n] <> C[n]) AND (C[n] <> 0)) OR CountTrip[n]) ;Use for Bag Arrived at destination
	CountOld[n] 	= C[n]

ENDLOOP
END_PROGRAM
```

### Program Logical/Sequences/zzbagsfl (IEC, version 1.00.0) - * Bag Shuffle including Buffers - Using 'Bag' 

#### zzbagsflCyclic.ab
```automation-basic
PROGRAM _CYCLIC
	(* cyclic program *)

;-----------------------------------------------------------
;Revision 1.00 19/12/2005 D.J. First Issue - Using BAG array
;-----------------------------------------------------------

Std.BagsWithDestinations 	= FALSE
Std.CustomerFound	 		= FALSE

LOOP CurrentLine = 1 to Std.MaxLinesBuffers DO

	LineSp = 0

	LOOP CurrentBag = Line[CurrentLine].FirstBag  TO Line[CurrentLine].LastBag DO

		EXITIF Line[CurrentLine].FirstBag = 0

		NextBag = (CurrentBag + 1)

		IF ((CurrentBag < Line[CurrentLine].LastBag) AND ((Bag[CurrentBag].Cat = 0) AND (Bag[NextBag].Cat > 0))) THEN

			;Copy Next Bag to Current
			Bag[CurrentBag]	= Bag[NextBag]
			Bag[NextBag] 	= Bag[0]

		ENDIF

		IF ((Bag[CurrentBag].Dst > 0) AND (CurrentLine <= Std.MaxLines)) THEN
			Std.BagsWithDestinations = TRUE
		ENDIF

		;Add the line spaces up
		IF Bag[CurrentBag].Cat = 0 THEN
			LineSp = (LineSp + 1)
		ENDIF

		;For Customer FIFO table
		;-----------------------
		;Customer at front of FIFO in Storage
		IF ((Bag[CurrentBag].Cus = D[401]) AND (D[401] > 0) AND (CurrentLine <= Std.MaxLines)) THEN
			Std.CustomerFound	 	= TRUE
		ENDIF

	ENDLOOP
	;Save the number of spaces on the current line
	Line[CurrentLine].Space = LineSp

ENDLOOP

END_PROGRAM
```

### Program Logical/Sequences/zzbitcal (IEC, version 3.00.0) - * Bags In Transit Calculation

#### zzbitcal.var
```iecst
VAR RETAIN
	TotalTransitBags	:UINT;
	n	:UINT;
	BITDest	:ARRAY [0..99] OF UINT;
	Destination	:USINT;
	SpaceBIT	:ARRAY [0..99] OF UINT;
	Spaces	:INT;
END_VAR

VAR
	BITBag	:UINT;
END_VAR
```

#### zzbitcalInit.ab
```automation-basic
PROGRAM _INIT
	(* init program *)

BITBag = 1

;Transfer Belt Bags - Pair loop
LOOP n = 200 TO 226 DO
	BITDest[BITBag] = n
	BITBag = BITBag + 1
ENDLOOP

;Bags in transit
;LOOP n = 140 to 179 DO
	;BITDest[BITBag] = n
	;BITBag = BITBag + 1
;ENDLOOP

TotalTransitBags = (BITBag - 1)
END_PROGRAM
```

### Program Logical/Sequences/zcusfifo (IEC, version 2.10.0) - * Customer FIFO 

#### zcusfifoCyclic.ab
```automation-basic
PROGRAM _CYCLIC
;------------------------------------------------------
;Revision 1.00 11/02/2002 D.J. First Issue
;Revision 2.00 11/06/2002 D.J. Included Bags In Transit
;------------------------------------------------------

;Include any Bags In Transit if required

;Check if found in Bags in transit
;IF (Bag[104].Cus = D[401]) AND (D[401] > 0)) THEN		;Offgoing BIT
;	Std.CustomerFound = TRUE
;ENDIF
;IF (Bag[105].Cus = D[401]) AND (D[401] > 0)) THEN		;SIC1 Bag
;	Std.CustomerFound = TRUE
;ENDIF
;IF (Bag[106].Cus = D[401]) AND (D[401] > 0)) THEN		;Pairing Loop BIT
;	Std.CustomerFound = TRUE
;ENDIF

;New Customers
OngoingCus 	= D[498]
EditCus		= D[499]

IF Std.CustomerFIFO THEN

	;The following are Set by the "Bag Shuffle"
	;First customer not found clear from the FIFO
	IF NOT Std.CustomerFound THEN
		D[401] = 0
	ENDIF

	;Shuffle the Table down
	D[400] = 0

	LOOP n = 401 TO 496 DO

		IF ((D[n] = 0) AND (D[n + 1] > 0)) THEN
			D[n] = D[n + 1]
			D[n + 1] = 0
		ENDIF

		IF (D[n] > 0) THEN
			;Inc FIFO Header Count
			D[400] = (D[400] + 1)
		ENDIF

		;Clear New Customer if found
		IF ((OngoingCus > 0) AND (OngoingCus = D[n])) THEN
			OngoingCus = 0
		ENDIF

		;Clear Edited Customer if found
		IF ((EditCus > 0) AND (EditCus = D[n])) THEN
			EditCus = 0
		ENDIF

	ENDLOOP

	;D498 = Ongoing New Customer
	IF ((OngoingCus > 0) AND (D[401 + D[400]] = 0)) THEN
		D[401 + D[400]]	= OngoingCus
		OngoingCus 		= 0
		D[400] 			= (D[400] + 1)
	ENDIF

	;D499 = Edited New Customer
	IF ((EditCus > 0) AND (D[401 + D[400]] = 0)) THEN
		D[401 + D[400]]	= EditCus
		EditCus 		= 0
		D[400] 			= (D[400] + 1)
	ENDIF

	;Find the Current Customer for each Discharger and allocate the Next Customer

	LOOP x = 1 TO Std.MaxDischargers DO

		Uld[x].FIFONextCustomer = 0
		Uld[x].FIFOCustomerFound = FALSE

		;If No Customer then Allocate with the First
		IF (Uld[x].FIFOCustomer = 0) THEN
			Uld[x].FIFOCustomer = D[401]
		ENDIF

		;If Next Customer available then allocate New Customer
		IF (D[400] > 0) THEN
			LOOP n = 401 TO (D[400] + 400) DO
				IF ((Uld[x].FIFOCustomer = D[n]) AND (D[n] > 0)) THEN
					Uld[x].FIFOCustomerFound = TRUE
					IF (D[n + 1] > 0) THEN
						Uld[x].FIFONextCustomer = D[n + 1]
					ENDIF
				ENDIF
			ENDLOOP
		ENDIF

		;If the current customer has been removed then set the next as the first
		IF ((Uld[x].FIFONextCustomer = 0) AND NOT Uld[x].FIFOCustomerFound) THEN
			Uld[x].FIFONextCustomer = D[401]
		ENDIF

	ENDLOOP

ENDIF

D[498] = OngoingCus
D[499] = EditCus
END_PROGRAM
```

### Program Logical/Sequences/zztcpip (IEC) - * TCP IP Communications

#### zztcpip.var
```iecst
VAR
	Port	:UINT;
	IPAddr	:UDINT;
	TCPsend_1	:TCPsend;
	TCPserv_1	:TCPserv;
	NoDataET	:TIME;
	NoData	:BOOL;
	PLS	:BOOL;
	RXStatus	:UINT;
	TCPclose_1	:TCPclose;
	RXLength	:UDINT;
	NEWSTEP	:UINT;
	STEP	:UINT;
	TCPrecv_1	:TCPrecv;
	rdata	:ARRAY [0..1023] OF USINT;
	Data_Array_Type	:INT;
	Data_array_adr	:UDINT;
	Data_StartH	:UINT;
	Data_Start	:UINT;
	Data_Amount	:UINT;
	Data_Valid	:BOOL;
	Data_RXTX_Type	:INT;
	LengthValid	:BOOL;
	tx_frame	:ARRAY [0..2047] OF USINT;
	WriteEnable	:BOOL;
	tx_length	:UINT;
	RXValid	:UINT;
	Data_AmountH	:UINT;
	NEWSTEP2	:UINT;
	STEP2	:UINT;
	TCPserv_2	:TCPserv;
	Port2	:UINT;
	IPAddr2	:UDINT;
	PLS2	:BOOL;
	WriteEnable2	:BOOL;
	TCPsend_2	:TCPsend;
	TCPrecv_2	:TCPrecv;
	rdata2	:ARRAY [0..1023] OF USINT;
	RXLength2	:UDINT;
	RXStatus2	:UINT;
	RXValid2	:UINT;
	tx_frame2	:ARRAY [0..2047] OF USINT;
	tx_length2	:UINT;
	NoData2	:BOOL;
	NoData2ET	:TIME;
	TCPclose_2	:TCPclose;
	PacketID	:USINT;
	EnableConnection1	:BOOL;
	EnableConnection2	:BOOL;
	ResetConnection	:BOOL;
END_VAR
```

#### zztcpipInit.ab
```automation-basic
PROGRAM _INIT
(* init program *)

;Enable connections set to TRUE or FALSE depending on how many connections are required
EnableConnection1 = TRUE
EnableConnection2 = TRUE

;Start Connection
ResetConnection = TRUE
END_PROGRAM
```

### Program Logical/Sequences/zzforceo (IEC, version 1.00.0) - * PLC Output forcing from graphics

#### zzforceoInit.ab
```automation-basic
PROGRAM _INIT
(* init program *)

;Clear force registers

D[303] = 0
D[304] = 0
D[305] = 0

;Clear force disable
memset(ADR(YForceDisable),0, SIZEOF(YForceDisable))
END_PROGRAM
```

### Program Logical/Sequences/zzuld_3 (IEC, version 1.00.0) - * Unloading 3
